       #sTimerLoadGripperOpened(IN := #sCurrent_Step_NB = 90 AND #iLoadGripperOpened,
                                PT := T#200ms);

       // Timer between approach and Load position
       #sTimerAfterApproach(IN := #sCurrent_Step_NB = 75 AND #iAxisW_FixtApproachPos,
                            PT := T#100ms);
   END_REGION

   REGION Sequence Function
       CASE #sCurrent_Step_NB OF
           #S00_INIT:
               REGION S00 INIT
                   #sCheck_Step_Condition := TRUE;
               END_REGION
           #S10_CHECK_FIXTURE_LOAD_OPTION:
               REGION S10_CHECK_FIXTURE_LOAD_OPTION
                   #sCheck_Step_Condition := TRUE;
               END_REGION
           #S20_AXIS_W_TO_FIXTURE_SAFE_POS_START_REQ:
               REGION S20_AXIS_W_TO_FIXTURE_SAFE_POS_START_REQ
                   #sAxisW_StartReq := NOT #iAxisW_FixtSafePos;
                   #sAxisW_PosSetPoint := LREAL_TO_REAL(#iAxisW_FixtSafePosSetPoint);
                   #sCheck_Step_Condition := TRUE;
               END_REGION
           #S30_AXIS_W_TO_FIXTURE_SAFE_POS_REACHED:
               REGION S30_AXIS_W_TO_FIXTURE_SAFE_POS_REACHED
                   #sCheck_Step_Condition := TRUE;
               END_REGION
           #S40_AXIS_V_TO_FIXTURE_LOAD_POS_START_REQ:
               REGION S40_AXIS_V_TO_FIXTURE_LOAD_POS_START_REQ
                   #sAxisV_StartReq := NOT #iAxisV_FixtLoadPos;
                   #sAxisV_PosSetPoint := LREAL_TO_REAL(#iAxisV_FixtLoadPosSetPoint);
                   #sCheck_Step_Condition := TRUE;
               END_REGION
           #S50_AXIS_V_TO_FIXTURE_LOAD_POS_REACHED:
               REGION S50_AXIS_V_TO_FIXTURE_LOAD_POS_REACHED
                   #sCheck_Step_Condition := TRUE;
               END_REGION
           #S60_OPEN_FIXTURE:
               REGION S60_OPEN_FIXTURE
                   #sFixtureOpenReq := TRUE;
                   IF #sTimerFixtureOpened.Q THEN
                       #sCheck_Step_Condition := TRUE;
                   END_IF;
               END_REGION


           #S70_AXIS_W_TO_FIXTURE_APPROACH_POS_START_REQ:
               REGION S70_AXIS_W_TO_FIXTURE_APPROACH_POS_START_REQ
                   #sAxisW_StartReq := NOT #iAxisW_FixtApproachPos;
                   #sAxisW_PosSetPoint := LREAL_TO_REAL(#iAxisW_FixtApproachPosSetPoint);
                   #sCheck_Step_Condition := TRUE;
               END_REGION
           #S75_AXIS_W_TO_FIXTURE_APPROACH_POS_REACHED:
               REGION S75_AXIS_W_TO_FIXTURE_APPROACH_POS_REACHED
                   IF #sTimerAfterApproach.Q THEN
                       #sCheck_Step_Condition := TRUE;
                   END_IF;
               END_REGION


           #S80_AXIS_W_TO_FIXTURE_LOAD_POS_START_REQ:
               REGION #S80_AXIS_W_TO_FIXTURE_LOAD_POS_START_REQ
                   #sAxisW_StartReq := NOT #iAxisW_FixtLoadPos;
                   #sAxisW_PosSetPoint := LREAL_TO_REAL(#iAxisW_FixtLoadPosSetPoint);
                   #sCheck_Step_Condition := TRUE;
               END_REGION
           #S85_AXIS_W_TO_FIXTURE_LOAD_POS_REACHED:
               REGION #S85_AXIS_W_TO_FIXTURE_LOAD_POS_REACHED
                   #sCheck_Step_Condition := TRUE;
               END_REGION
           #S90_OPEN_LOAD_GRIPPER:
               REGION S90_OPEN_LOAD_GRIPPER
                   #sLoadGripperOpenReq := TRUE;
                   IF #sTimerLoadGripperOpened.Q THEN
                       #sCheck_Step_Condition := TRUE;
                   END_IF;
               END_REGION
           #S95_VACUUM_START:
               REGION S95_VACUUM_START
                   #sVacuumStartReq := TRUE;
                   #sCheck_Step_Condition := TRUE;
               END_REGION
           #S100_AXIS_W_TO_FIXTURE_SAFE_POS_START_REQ:
               REGION S100_AXIS_W_TO_FIXTURE_SAFE_POS_START_REQ
                   #sAxisW_StartReq := NOT #iAxisW_FixtSafePos;
                   #sAxisW_PosSetPoint := LREAL_TO_REAL(#iAxisW_FixtSafePosSetPoint);
                   #sCheck_Step_Condition := TRUE;
               END_REGION
           #S110_AXIS_W_TO_FIXTURE_SAFE_POS_REACHED:
               REGION S110_AXIS_W_TO_FIXTURE_SAFE_POS_REACHED
                   #sCheck_Step_Condition := TRUE;
               END_REGION
           #S120_CLOSE_FIXTURE:
               REGION S120_CLOSE_FIXTURE
                   #sFixtureCloseReq := TRUE;
                   IF #sTimerFixtureClosed.Q THEN
                       #sCheck_Step_Condition := TRUE;
                   END_IF;
               END_REGION
           #S195_JOB_DONE:
               REGION S195_JOB_DONE
                   #sInterface.JobDone := TRUE;
                   #sCheck_Step_Condition := TRUE;
               END_REGION
           ELSE:
               #sInterface.Error := TRUE;
       END_CASE;
   END_REGION

   REGION Sequence Next Step Condition
       IF #sCheck_Step_Condition THEN
           CASE #sCurrent_Step_NB OF
               #S00_INIT:
                   REGION S00_INIT
                       IF #sInterface.SequenceReleased AND #iJobReq THEN
                           #sCurrent_Step_NB := #S10_CHECK_FIXTURE_LOAD_OPTION;
                           #sInterface.SequenceRun := TRUE;
                           #sCheck_Step_Condition := FALSE;
                       ELSE
                           #sInterface.SequenceRun := FALSE;
                       END_IF;
                   END_REGION
               #S10_CHECK_FIXTURE_LOAD_OPTION:
                   REGION S10_CHECK_FIXTURE_LOAD_OPTION
                       IF #sInterface.SequenceReleased AND #sStepForward AND NOT "DB_LoaderOptions".Fixture.LoadingDisabled THEN
                           #sCurrent_Step_NB := #S20_AXIS_W_TO_FIXTURE_SAFE_POS_START_REQ;
                           #sCheck_Step_Condition := FALSE;
                       ELSIF #sInterface.SequenceReleased AND #sStepForward AND "DB_LoaderOptions".Fixture.LoadingDisabled THEN
                           #sCurrent_Step_NB := #S195_JOB_DONE;
                           #sCheck_Step_Condition := FALSE;
                       END_IF;
                   END_REGION
               #S20_AXIS_W_TO_FIXTURE_SAFE_POS_START_REQ:
                   REGION S20_AXIS_W_TO_FIXTURE_SAFE_POS_START_REQ
                       IF #sInterface.SequenceReleased AND #sStepForward AND (#iAxisW_Moving OR #iAxisW_FixtSafePos) THEN
                           #sCurrent_Step_NB := #S30_AXIS_W_TO_FIXTURE_SAFE_POS_REACHED;
                           #sCheck_Step_Condition := FALSE;
                       END_IF;
                   END_REGION
               #S30_AXIS_W_TO_FIXTURE_SAFE_POS_REACHED:
                   REGION S30_AXIS_W_TO_FIXTURE_SAFE_POS_REACHED
                       IF #sInterface.SequenceReleased AND #sStepForward AND NOT #sAxisW_StartReq AND #iAxisW_FixtSafePos THEN
                           #sCurrent_Step_NB := #S40_AXIS_V_TO_FIXTURE_LOAD_POS_START_REQ;
                           #sCheck_Step_Condition := FALSE;
                       END_IF;
                   END_REGION
               #S40_AXIS_V_TO_FIXTURE_LOAD_POS_START_REQ:
                   REGION S40_AXIS_V_TO_FIXTURE_LOAD_POS_START_REQ
                       IF #sInterface.SequenceReleased AND #sStepForward AND (#iAxisV_Moving OR #iAxisV_FixtLoadPos) THEN
                           #sCurrent_Step_NB := #S50_AXIS_V_TO_FIXTURE_LOAD_POS_REACHED;
                           #sCheck_Step_Condition := FALSE;
                       END_IF;
                   END_REGION
               #S50_AXIS_V_TO_FIXTURE_LOAD_POS_REACHED:
                   REGION S50_AXIS_V_TO_FIXTURE_LOAD_POS_REACHED
                       IF #sInterface.SequenceReleased AND #sStepForward AND NOT #sAxisV_StartReq AND #iAxisV_FixtLoadPos THEN
                           #sCurrent_Step_NB := #S60_OPEN_FIXTURE;
                           #sCheck_Step_Condition := FALSE;
                       END_IF;
                   END_REGION
               #S60_OPEN_FIXTURE:
                   REGION S60_OPEN_FIXTURE
                       IF #sInterface.SequenceReleased AND #sStepForward AND #iFixtureOpened THEN
                           #sCurrent_Step_NB := #S70_AXIS_W_TO_FIXTURE_APPROACH_POS_START_REQ;
                           #sCheck_Step_Condition := FALSE;
                       END_IF;
                   END_REGION
               #S70_AXIS_W_TO_FIXTURE_APPROACH_POS_START_REQ:
                   REGION S70_AXIS_W_TO_FIXTURE_APPROACH_POS_START_REQ
                       IF #sInterface.SequenceReleased AND #sStepForward AND (#iAxisW_Moving OR #iAxisW_FixtApproachPos) THEN
                           #sCurrent_Step_NB := #S75_AXIS_W_TO_FIXTURE_APPROACH_POS_REACHED;
                           #sCheck_Step_Condition := FALSE;
                       END_IF;
                   END_REGION
               #S75_AXIS_W_TO_FIXTURE_APPROACH_POS_REACHED:
                   REGION S75_AXIS_W_TO_FIXTURE_APPROACH_POS_REACHED
                       IF #sInterface.SequenceReleased AND #sStepForward AND NOT #sAxisW_StartReq AND #iAxisW_FixtApproachPos THEN
                           #sCurrent_Step_NB := #S80_AXIS_W_TO_FIXTURE_LOAD_POS_START_REQ;
                           #sCheck_Step_Condition := FALSE;
                       END_IF;
                   END_REGION

               #S80_AXIS_W_TO_FIXTURE_LOAD_POS_START_REQ:
                   REGION S80_AXIS_W_TO_FIXTURE_LOAD_POS_START_REQ
                       IF #sInterface.SequenceReleased AND #sStepForward AND (#iAxisW_Moving OR #iAxisW_FixtLoadPos) THEN
                           #sCurrent_Step_NB := #S85_AXIS_W_TO_FIXTURE_LOAD_POS_REACHED;
                           #sCheck_Step_Condition := FALSE;
                       END_IF;
                   END_REGION
               #S85_AXIS_W_TO_FIXTURE_LOAD_POS_REACHED:
                   REGION S85_AXIS_W_TO_FIXTURE_LOAD_POS_REACHED
                       IF #sInterface.SequenceReleased AND #sStepForward AND NOT #sAxisW_StartReq AND #iAxisW_FixtLoadPos THEN
                           #sCurrent_Step_NB := #S90_OPEN_LOAD_GRIPPER;
                           #sCheck_Step_Condition := FALSE;
                       END_IF;
                   END_REGION


               #S90_OPEN_LOAD_GRIPPER:
                   REGION S90_OPEN_LOAD_GRIPPER
                       IF #sInterface.SequenceReleased AND #sStepForward AND #iLoadGripperOpened THEN
                           #sCurrent_Step_NB := #S95_VACUUM_START;
                           #sCheck_Step_Condition := FALSE;
                       END_IF;
                   END_REGION
               #S95_VACUUM_START:
                   REGION S95_VACUUM_START
                       IF #sInterface.SequenceReleased AND #sStepForward AND TRUE THEN
                           #sCurrent_Step_NB := #S100_AXIS_W_TO_FIXTURE_SAFE_POS_START_REQ;
                           #sCheck_Step_Condition := FALSE;
                       END_IF;
                   END_REGION
               #S100_AXIS_W_TO_FIXTURE_SAFE_POS_START_REQ:
                   REGION S100_AXIS_W_TO_FIXTURE_SAFE_POS_START_REQ
                       IF #sInterface.SequenceReleased AND #sStepForward AND (#iAxisW_Moving OR #iAxisW_FixtSafePos) THEN
                           #sCurrent_Step_NB := #S110_AXIS_W_TO_FIXTURE_SAFE_POS_REACHED;
                           #sCheck_Step_Condition := FALSE;
                       END_IF;
                   END_REGION
               #S110_AXIS_W_TO_FIXTURE_SAFE_POS_REACHED:
                   REGION S110_AXIS_W_TO_FIXTURE_SAFE_POS_REACHED
                       IF #sInterface.SequenceReleased AND #sStepForward AND NOT #sAxisW_StartReq AND #iAxisW_FixtSafePos THEN
                           #sCurrent_Step_NB := #S120_CLOSE_FIXTURE;
                           #sCheck_Step_Condition := FALSE;
                       END_IF;
                   END_REGION
               #S120_CLOSE_FIXTURE:
                   REGION S120_CLOSE_FIXTURE
                       IF #sInterface.SequenceReleased AND #sStepForward AND #iFixtureClosed THEN
                           #sCurrent_Step_NB := #S195_JOB_DONE;
                           #sCheck_Step_Condition := FALSE;
                       END_IF;
                   END_REGION
               #S195_JOB_DONE:
                   REGION S195_JOB_DONE
                       IF NOT #iJobReq THEN
                           #sCurrent_Step_NB := #S00_INIT;
                           #sCheck_Step_Condition := FALSE;
                           #sInterface.JobDone := FALSE;
                       END_IF;
                   END_REGION
               ELSE
                   #sInterface.Error := TRUE;
           END_CASE;
       END_IF;
   END_REGION

   REGION Outputs Update
       #oAxisV_StartReq := #sAxisV_StartReq;
       #oAxisV_PosSetPoint := #sAxisV_PosSetPoint;
       #oAxisW_StartReq := #sAxisW_StartReq;
       #oAxisW_PosSetPoint := #sAxisW_PosSetPoint;
       #oFixtureOpenReq := #sFixtureOpenReq;
       #oFixtureCloseReq := #sFixtureCloseReq;
       #oLoadGripperOpenReq := #sLoadGripperOpenReq;
       #oVacuumStartReq := #sVacuumStartReq;
   END_REGION

   REGION Steps - Date and Time History
       IF #sHistory.Activation THEN
           IF #sHistory.Steps[0] <> #sCurrent_Step_NB THEN
               FOR #tIndex := 98 TO 0 BY -1 DO
                   #sHistory.Steps[#tIndex + 1] := #sHistory.Steps[#tIndex];
                   #sHistory.Date_Time[#tIndex + 1] := #sHistory.Date_Time[#tIndex];
               END_FOR;
               #sHistory.Steps[0] := #sCurrent_Step_NB;
               #sHistory.Date_Time[0] := #iPLC_DateAndTime;
           END_IF;
       END_IF;
   END_REGION

   REGION Steps Text
       #StepText(iErrorCode := #sCurrent_Step_NB,
                 oErrorText => #StepText.oErrorText);
   END_REGION
END_FUNCTION_BLOCK

FUNCTION_BLOCK "FB_FixtureBlowing"   // FB68, SCL
{ S7_Optimized_Access := 'TRUE' }
// stored: AutoNumber false, MemoryReserve 100, SetENOAutomatically false
   VAR_INPUT
      iStartSeqCond : Bool;   // Start Sequence Conditions
      iJobReq : Bool;   // Job Request - From Main
      iFixtureOpened : Bool;
      iAxisV_FixtBlowingPos : Bool;
      iAxisV_FixtBlowingPosSetPoint : LReal;
      iAxisW_FixtSafePos : Bool;
      iAxisW_FixtSafePosSetPoint : LReal;
      iAxisW_FixtBlowPos : Bool;
      iAxisW_FixtBlowPosSetPoint : LReal;
      iAxisV_Moving : Bool;   // Shuttle is moving
      iAxisV_InPos : Bool;
      iAxisW_Moving { ExternalAccessible := 'False'; ExternalVisible := 'False'; ExternalWritable := 'False'} : Bool;   // Shuttle is moving
      iAxisW_InPos : Bool;
      iBlowingTime : Time;
      iPLC_DateAndTime : DTL;
      iStepPause : Bool;
   END_VAR
   VAR_OUTPUT
      oFixtureOpenReq : Bool;
      oAxisV_StartReq : Bool;
      oAxisV_PosSetPoint : Real;
      oAxisW_StartReq : Bool;
      oAxisW_PosSetPoint : Real;
      oBlowingReq : Bool;
   END_VAR
   VAR
      sCurrent_Step_NB : Int;   // Active Step Number
      sCheck_Step_Condition : Bool;
      sOneStepForward : Bool;
      sRTOneStepForward : R_TRIG;
      sOneStepMode { S7_SetPoint := 'True'} : Bool;
      sStepForward : Bool;
      sInterface : "UDT_SequenceInterface";
      sFixtureOpenReq { S7_SetPoint := 'True'} : Bool;
      sAxisV_StartReq : Bool;
      sAxisV_PosSetPoint : Real;
      sAxisW_StartReq : Bool;
      sAxisW_PosSetPoint : Real;
      sBlowingReq : Bool;   // Drilled Part To Unload - From FB_Position
      sBlowingTimerStart : Bool;
      sBlowingTimer : TP_TIME;
      sFT_BlowingTimer { S7_SetPoint := 'True'} : F_TRIG;
      sTimerFixtureOpened : TON_TIME;
      sHistory : Struct
         Activation : Bool;
         Steps : Array[0..99] of Int;
         Date_Time : Array[0..99] of DTL;
      END_STRUCT;
      StepText : "FB_GetTextErrorCode";
   END_VAR
   VAR_TEMP
      tIndex : Int;   // Index
   END_VAR
   VAR CONSTANT
      S00_INIT : Int := 0;
      S10_CHECK_FIXTURE_BLOW_OPTION : Int := 10;
      S20_AXIS_W_TO_FIXTURE_SAFE_POS_START_REQ : Int := 20;
      S30_AXIS_W_TO_FIXTURE_SAFE_POS_REACHED : Int := 30;
      S40_AXIS_V_TO_FIXTURE_BLOW_POS_START_REQ : Int := 40;
      S50_AXIS_V_TO_FIXTURE_BLOW_POS_REACHED : Int := 50;
      S60_OPEN_FIXTURE : Int := 60;
      S70_AXIS_W_TO_FIXTURE_BLOW_POS_START_REQ : Int := 70;
      S80_AXIS_W_TO_FIXTURE_BLOW_POS_REACHED : Int := 80;
      S90_BLOWING_TIMER_START_REQ : Int := 90;
      S100_AXIS_W_TO_FIXTURE_SAFE_POS_START_REQ : Int := 100;
      S110_AXIS_W_TO_FIXTURE_SAFE_POS_REACHED : Int := 110;
      S195_JOB_DONE : Int := 195;
   END_VAR
   // StepText.sCode_error[0].ErrorCode := 0;
   // StepText.sCode_error[1].ErrorCode := 10;
   // StepText.sCode_error[2].ErrorCode := 20;
   // StepText.sCode_error[3].ErrorCode := 30;
   // StepText.sCode_error[4].ErrorCode := 40;
   // StepText.sCode_error[5].ErrorCode := 50;
   // StepText.sCode_error[6].ErrorCode := 60;
   // StepText.sCode_error[7].ErrorCode := 70;
   // StepText.sCode_error[8].ErrorCode := 80;
   // StepText.sCode_error[9].ErrorCode := 90;
   // StepText.sCode_error[10].ErrorCode := 95;
BEGIN
   REGION Description header 
       //==================================================================================
       // POSALUX Swiss SA / (C) Copyright 2026
       //----------------------------------------------------------------------------------
       // Title: FB_FixtureBlowing
       // Comment/Function: 
       // Author: Fabien WALDT
       // Engineering: TIA Portal v20
       //----------------------------------------------------------------------------------
       // Change log table:
       // Version  | Date     | Expert in charge | Changes applied
       // ---------|----------|------------------|-----------------------------------------
       // 00.00.01 | 20260122 | WFA              | First released version
       // =================================================================================
   END_REGION

   REGION Define condition to start
       IF #iStartSeqCond THEN
           #sInterface.SequenceReleased := TRUE;
       ELSE
           // Standard sequencer controls
           #sInterface.SequenceReleased := FALSE;
           #sCurrent_Step_NB := #S00_INIT;
           #sInterface.SequenceRun := FALSE;
           #sInterface.JobDone := FALSE;
           #sCheck_Step_Condition := FALSE;

           // Dedicated sequencer controls
           #sAxisV_StartReq := FALSE;
           #sAxisV_PosSetPoint := 0.0;
           #sAxisW_StartReq := FALSE;
           #sAxisW_PosSetPoint := 0.0;
           #sFixtureOpenReq := FALSE;
           #sBlowingReq := FALSE;
           #sBlowingTimerStart := FALSE;

           // Add specifics controls 
       END_IF;

       // Reset interface error
       IF #sInterface.Reset THEN
           #sInterface.Error := FALSE;
       END_IF;

       // Reset start when axis in position
       IF #iAxisV_InPos THEN
           #sAxisV_StartReq := FALSE;
       END_IF;
       IF #iAxisW_InPos THEN
           #sAxisW_StartReq := FALSE;
       END_IF;

       // One step forward
       #sRTOneStepForward.CLK := #sOneStepForward;
       #sRTOneStepForward();
       #sStepForward := (NOT #sOneStepMode OR (#sOneStepMode AND #sRTOneStepForward.Q)) AND NOT #iStepPause;
       #sOneStepForward := FALSE;

       // Blowing Timer
       #sBlowingTimer(IN := #sBlowingTimerStart,
                      PT := #iBlowingTime);

       #sFT_BlowingTimer(CLK := #sBlowingTimer.Q);

       #sBlowingReq := #sBlowingTimer.Q
       OR #sCurrent_Step_NB = 70
       OR #sCurrent_Step_NB = 80;
       // Action only true in dedicated steps
       #sFixtureOpenReq := FALSE;
       #sBlowingTimerStart := FALSE;

       // Step Timer
       #sTimerFixtureOpened(IN := #sCurrent_Step_NB = 60 AND #iFixtureOpened,
                            PT := T#1000ms);
   END_REGION

   REGION Sequence Function
       CASE #sCurrent_Step_NB OF
           #S00_INIT:
               REGION S00 INIT
                   #sCheck_Step_Condition := TRUE;
               END_REGION
           #S10_CHECK_FIXTURE_BLOW_OPTION:
               REGION S10_CHECK_FIXTURE_BLOW_OPTION
                   #sCheck_Step_Condition := TRUE;
               END_REGION
           #S20_AXIS_W_TO_FIXTURE_SAFE_POS_START_REQ:
               REGION S20_AXIS_W_TO_FIXTURE_SAFE_POS_START_REQ
                   #sAxisW_StartReq := NOT #iAxisW_FixtSafePos;
                   #sAxisW_PosSetPoint := LREAL_TO_REAL(#iAxisW_FixtSafePosSetPoint);
                   #sCheck_Step_Condition := TRUE;
               END_REGION
           #S30_AXIS_W_TO_FIXTURE_SAFE_POS_REACHED:
               REGION S30_AXIS_W_TO_FIXTURE_SAFE_POS_REACHED
                   #sCheck_Step_Condition := TRUE;
               END_REGION
           #S40_AXIS_V_TO_FIXTURE_BLOW_POS_START_REQ:
               REGION S40_AXIS_V_TO_FIXTURE_BLOW_POS_START_REQ
                   #sAxisV_StartReq := NOT #iAxisV_FixtBlowingPos;
                   #sAxisV_PosSetPoint := LREAL_TO_REAL(#iAxisV_FixtBlowingPosSetPoint);
                   #sCheck_Step_Condition := TRUE;
               END_REGION
           #S50_AXIS_V_TO_FIXTURE_BLOW_POS_REACHED:
               REGION S50_AXIS_V_TO_FIXTURE_BLOW_POS_REACHED
                   #sCheck_Step_Condition := TRUE;
               END_REGION
           #S60_OPEN_FIXTURE:
               REGION S60_OPEN_FIXTURE
                   #sFixtureOpenReq := TRUE;
                   IF #sTimerFixtureOpened.Q THEN
                       #sCheck_Step_Condition := TRUE;
                   END_IF;
               END_REGION
           #S70_AXIS_W_TO_FIXTURE_BLOW_POS_START_REQ:
               REGION S70_AXIS_W_TO_FIXTURE_BLOW_POS_START_REQ
                   #sAxisW_StartReq := NOT #iAxisW_FixtBlowPos;
                   #sAxisW_PosSetPoint := LREAL_TO_REAL(#iAxisW_FixtBlowPosSetPoint);
                   #sCheck_Step_Condition := TRUE;
               END_REGION
           #S80_AXIS_W_TO_FIXTURE_BLOW_POS_REACHED:
               REGION S80_AXIS_W_TO_FIXTURE_BLOW_POS_REACHED
                   #sCheck_Step_Condition := TRUE;
               END_REGION
           #S90_BLOWING_TIMER_START_REQ:
               REGION S90_BLOWING_TIMER_START_REQ
                   #sBlowingTimerStart := TRUE;
                   #sCheck_Step_Condition := TRUE;
               END_REGION
           #S100_AXIS_W_TO_FIXTURE_SAFE_POS_START_REQ:
               REGION S100_AXIS_W_TO_FIXTURE_SAFE_POS_START_REQ
                   #sAxisW_StartReq := NOT #iAxisW_FixtSafePos;
                   #sAxisW_PosSetPoint := LREAL_TO_REAL(#iAxisW_FixtSafePosSetPoint);
                   #sCheck_Step_Condition := TRUE;
               END_REGION
           #S110_AXIS_W_TO_FIXTURE_SAFE_POS_REACHED:
               REGION S110_AXIS_W_TO_FIXTURE_SAFE_POS_REACHED
                   #sCheck_Step_Condition := TRUE;
               END_REGION
           #S195_JOB_DONE:
               REGION S195_JOB_DONE
                   #sInterface.JobDone := TRUE;
                   #sCheck_Step_Condition := TRUE;
               END_REGION
           ELSE:
               #sInterface.Error := TRUE;
       END_CASE;
   END_REGION

   REGION Sequence Next Step Condition
       IF #sCheck_Step_Condition THEN
           CASE #sCurrent_Step_NB OF
               #S00_INIT:
                   REGION S00_INIT
                       IF #sInterface.SequenceReleased AND #iJobReq THEN
                           #sCurrent_Step_NB := #S10_CHECK_FIXTURE_BLOW_OPTION;
                           #sInterface.SequenceRun := TRUE;
                           #sCheck_Step_Condition := FALSE;
                       ELSE
                           #sInterface.SequenceRun := FALSE;
                       END_IF;
                   END_REGION
               #S10_CHECK_FIXTURE_BLOW_OPTION:
                   REGION S10_CHECK_FIXTURE_UNLOAD_OPTION
                       IF #sInterface.SequenceReleased AND #sStepForward AND NOT "DB_LoaderOptions".Fixture.BlowingDisabled  THEN
                           #sCurrent_Step_NB := #S20_AXIS_W_TO_FIXTURE_SAFE_POS_START_REQ;
                           #sCheck_Step_Condition := FALSE;
                       ELSIF #sInterface.SequenceReleased AND #sStepForward AND "DB_LoaderOptions".Fixture.BlowingDisabled THEN
                           #sCurrent_Step_NB := #S195_JOB_DONE;
                           #sCheck_Step_Condition := FALSE;
                       END_IF;
                   END_REGION
               #S20_AXIS_W_TO_FIXTURE_SAFE_POS_START_REQ:
                   REGION S20_AXIS_W_TO_FIXTURE_SAFE_POS_START_REQ
                       IF #sInterface.SequenceReleased AND #sStepForward AND (#iAxisW_Moving OR #iAxisW_FixtSafePos) THEN
                           #sCurrent_Step_NB := #S30_AXIS_W_TO_FIXTURE_SAFE_POS_REACHED;
                           #sCheck_Step_Condition := FALSE;
                       END_IF;
                   END_REGION
               #S30_AXIS_W_TO_FIXTURE_SAFE_POS_REACHED:
                   REGION S30_AXIS_W_TO_FIXTURE_SAFE_POS_REACHED
                       IF #sInterface.SequenceReleased AND #sStepForward AND NOT #sAxisW_StartReq AND #iAxisW_FixtSafePos THEN
                           #sCurrent_Step_NB := #S40_AXIS_V_TO_FIXTURE_BLOW_POS_START_REQ;
                           #sCheck_Step_Condition := FALSE;
                       END_IF;
                   END_REGION
               #S40_AXIS_V_TO_FIXTURE_BLOW_POS_START_REQ:
                   REGION S40_AXIS_V_TO_FIXTURE_BLOW_POS_START_REQ
                       IF #sInterface.SequenceReleased AND #sStepForward AND (#iAxisV_Moving OR #iAxisV_FixtBlowingPos) THEN
                           #sCurrent_Step_NB := #S50_AXIS_V_TO_FIXTURE_BLOW_POS_REACHED;
                           #sCheck_Step_Condition := FALSE;
                       END_IF;
                   END_REGION
               #S50_AXIS_V_TO_FIXTURE_BLOW_POS_REACHED:
                   REGION S50_AXIS_V_TO_FIXTURE_BLOW_POS_REACHED
                       IF #sInterface.SequenceReleased AND #sStepForward AND NOT #sAxisV_StartReq AND #iAxisV_FixtBlowingPos THEN
                           #sCurrent_Step_NB := #S60_OPEN_FIXTURE;
                           #sCheck_Step_Condition := FALSE;
                       END_IF;
                   END_REGION
               #S60_OPEN_FIXTURE:
                   REGION S60_OPEN_FIXTURE
                       IF #sInterface.SequenceReleased AND #sStepForward AND #iFixtureOpened THEN
                           #sCurrent_Step_NB := #S70_AXIS_W_TO_FIXTURE_BLOW_POS_START_REQ;
                           #sCheck_Step_Condition := FALSE;
                       END_IF;
                   END_REGION
               #S70_AXIS_W_TO_FIXTURE_BLOW_POS_START_REQ:
                   REGION S70_AXIS_W_TO_FIXTURE_BLOW_POS_START_REQ
                       IF #sInterface.SequenceReleased AND #sStepForward AND (#iAxisW_Moving OR #iAxisW_FixtBlowPos) THEN
                           #sCurrent_Step_NB := #S80_AXIS_W_TO_FIXTURE_BLOW_POS_REACHED;
                           #sCheck_Step_Condition := FALSE;
                       END_IF;
                   END_REGION
               #S80_AXIS_W_TO_FIXTURE_BLOW_POS_REACHED:
                   REGION S80_AXIS_W_TO_FIXTURE_BLOW_POS_REACHED
                       IF #sInterface.SequenceReleased AND #sStepForward AND NOT #sAxisW_StartReq AND #iAxisW_FixtBlowPos THEN
                           #sCurrent_Step_NB := #S90_BLOWING_TIMER_START_REQ;
                           #sCheck_Step_Condition := FALSE;
                       END_IF;
                   END_REGION
               #S90_BLOWING_TIMER_START_REQ:
                   REGION S90_BLOWING_TIMER_START_REQ
                       IF #sInterface.SequenceReleased AND #sStepForward AND #sFT_BlowingTimer.Q THEN
                           #sCurrent_Step_NB := #S100_AXIS_W_TO_FIXTURE_SAFE_POS_START_REQ;
                           #sCheck_Step_Condition := FALSE;
                       END_IF;
                   END_REGION
               #S100_AXIS_W_TO_FIXTURE_SAFE_POS_START_REQ:
                   REGION S100_AXIS_W_TO_FIXTURE_SAFE_POS_START_REQ
                       IF #sInterface.SequenceReleased AND #sStepForward AND (#iAxisW_Moving OR #iAxisW_FixtSafePos) THEN
                           #sCurrent_Step_NB := #S110_AXIS_W_TO_FIXTURE_SAFE_POS_REACHED;
                           #sCheck_Step_Condition := FALSE;
                       END_IF;
                   END_REGION
               #S110_AXIS_W_TO_FIXTURE_SAFE_POS_REACHED:
                   REGION S110_AXIS_W_TO_FIXTURE_SAFE_POS_REACHED
                       IF #sInterface.SequenceReleased AND #sStepForward AND NOT #sAxisW_StartReq AND #iAxisW_FixtSafePos THEN
                           #sCurrent_Step_NB := #S195_JOB_DONE;
                           #sCheck_Step_Condition := FALSE;
                       END_IF;
                   END_REGION
               #S195_JOB_DONE:
                   REGION S195_JOB_DONE
                       IF NOT #iJobReq THEN
                           #sCurrent_Step_NB := #S00_INIT;
                           #sCheck_Step_Condition := FALSE;
                           #sInterface.JobDone := FALSE;
                       END_IF;
                   END_REGION
               ELSE
                   #sInterface.Error := TRUE;
           END_CASE;
       END_IF;
   END_REGION

   REGION Outputs Update
       #oAxisV_StartReq := #sAxisV_StartReq;
       #oAxisV_PosSetPoint := #sAxisV_PosSetPoint;
       #oAxisW_StartReq := #sAxisW_StartReq;
       #oAxisW_PosSetPoint := #sAxisW_PosSetPoint;
       #oFixtureOpenReq := #sFixtureOpenReq;
       #oBlowingReq := #sBlowingReq;
   END_REGION

   REGION Steps - Date and Time History
       IF #sHistory.Activation THEN
           IF #sHistory.Steps[0] <> #sCurrent_Step_NB THEN
               FOR #tIndex := 98 TO 0 BY -1 DO
                   #sHistory.Steps[#tIndex + 1] := #sHistory.Steps[#tIndex];
                   #sHistory.Date_Time[#tIndex + 1] := #sHistory.Date_Time[#tIndex];
               END_FOR;
               #sHistory.Steps[0] := #sCurrent_Step_NB;
               #sHistory.Date_Time[0] := #iPLC_DateAndTime;
           END_IF;
       END_IF;
   END_REGION

   REGION Steps Text
       #StepText(iErrorCode := #sCurrent_Step_NB,
                 oErrorText => #StepText.oErrorText);
   END_REGION
END_FUNCTION_BLOCK

FUNCTION_BLOCK "FB_FixtureRelease"   // FB70, SCL
{ S7_Optimized_Access := 'TRUE' }
// stored: AutoNumber false, MemoryReserve 100, SetENOAutomatically false
   VAR_INPUT
      iStartSeqCond : Bool;   // Start Sequence Conditions
      iJobReq : Bool;   // Job Request - From Main
      iAxisV_SafePos : Bool;
      iAxisV_SafePosSetPoint : LReal;
      iAxisW_FixtSafePos : Bool;
      iAxisW_FixtSafePosSetPoint : LReal;
      iAxisV_Moving : Bool;   // Shuttle is moving
      iAxisV_InPos : Bool;
      iAxisW_Moving { ExternalAccessible := 'False'; ExternalVisible := 'False'; ExternalWritable := 'False'} : Bool;   // Shuttle is moving
      iAxisW_InPos : Bool;
      iPLC_DateAndTime : DTL;
      iStepPause : Bool;
   END_VAR
   VAR_OUTPUT
      oAxisV_StartReq : Bool;
      oAxisV_PosSetPoint : Real;
      oAxisW_StartReq : Bool;
      oAxisW_PosSetPoint : Real;
   END_VAR
   VAR
      sCurrent_Step_NB : Int;   // Active Step Number
      sCheck_Step_Condition : Bool;
      sOneStepForward : Bool;
      sRTOneStepForward : R_TRIG;
      sOneStepMode { S7_SetPoint := 'True'} : Bool;
      sStepForward : Bool;
      sInterface : "UDT_SequenceInterface";
      sAxisV_StartReq : Bool;
      sAxisV_PosSetPoint : Real;
      sAxisW_StartReq : Bool;
      sAxisW_PosSetPoint : Real;
      sHistory : Struct
         Activation : Bool;
         Steps : Array[0..99] of Int;
         Date_Time : Array[0..99] of DTL;
      END_STRUCT;
      StepText : "FB_GetTextErrorCode";
   END_VAR
   VAR_TEMP
      tIndex : Int;   // Index
   END_VAR
   VAR CONSTANT
      S00_INIT : Int := 0;
      S10_CHECK_FIXTURE_RELEASE_OPTION : Int := 10;
      S20_AXIS_W_TO_FIXTURE_SAFE_POS_START_REQ : Int := 20;
      S30_AXIS_W_TO_FIXTURE_SAFE_POS_REACHED : Int := 30;
      S40_AXIS_V_TO_SHUTTLE_SAFE_POS_START_REQ : Int := 40;
      S50_AXIS_V_TO_SHUTTLE_SAFE_POS_REACHED : Int := 50;
      S95_JOB_DONE : Int := 95;
   END_VAR
   // StepText.sCode_error[0].ErrorCode := 0;
   // StepText.sCode_error[1].ErrorCode := 10;
   // StepText.sCode_error[2].ErrorCode := 20;
   // StepText.sCode_error[3].ErrorCode := 30;
   // StepText.sCode_error[4].ErrorCode := 40;
   // StepText.sCode_error[5].ErrorCode := 50;
   // StepText.sCode_error[6].ErrorCode := 60;
   // StepText.sCode_error[7].ErrorCode := 70;
   // StepText.sCode_error[8].ErrorCode := 80;
   // StepText.sCode_error[9].ErrorCode := 90;
   // StepText.sCode_error[10].ErrorCode := 95;
BEGIN
   REGION Description header 
       //==================================================================================
       // POSALUX Swiss SA / (C) Copyright 2026
       //----------------------------------------------------------------------------------
       // Title: FB_FixtureRelease
       // Comment/Function: 
       // Author: Fabien WALDT
       // Engineering: TIA Portal v20
       //----------------------------------------------------------------------------------
       // Change log table:
       // Version  | Date     | Expert in charge | Changes applied
       // ---------|----------|------------------|-----------------------------------------
       // 00.00.01 | 20260122 | WFA              | First released version
       // =================================================================================
   END_REGION

   REGION Define condition to start
       IF #iStartSeqCond THEN
           #sInterface.SequenceReleased := TRUE;
       ELSE
           // Standard sequencer controls
           #sInterface.SequenceReleased := FALSE;
           #sCurrent_Step_NB := #S00_INIT;
           #sInterface.SequenceRun := FALSE;
           #sInterface.JobDone := FALSE;
           #sCheck_Step_Condition := FALSE;

           // Dedicated sequencer controls
           #sAxisV_StartReq := FALSE;
           #sAxisV_PosSetPoint := 0.0;
           #sAxisW_StartReq := FALSE;
           #sAxisW_PosSetPoint := 0.0;

           // Add specifics controls 
       END_IF;

       // Reset interface error
       IF #sInterface.Reset THEN
           #sInterface.Error := FALSE;
       END_IF;

       // Reset start when axis in position
       IF #iAxisV_InPos THEN
           #sAxisV_StartReq := FALSE;
       END_IF;
       IF #iAxisW_InPos THEN
           #sAxisW_StartReq := FALSE;
       END_IF;

       // One step forward
       #sRTOneStepForward.CLK := #sOneStepForward;
       #sRTOneStepForward();
       #sStepForward := (NOT #sOneStepMode OR (#sOneStepMode AND #sRTOneStepForward.Q)) AND NOT #iStepPause;
       #sOneStepForward := FALSE;

       // Action only true in dedicated steps

       // Step Timer

   END_REGION

   REGION Sequence Function
       CASE #sCurrent_Step_NB OF
           #S00_INIT:
               REGION S00 INIT
                   #sCheck_Step_Condition := TRUE;
               END_REGION
           #S10_CHECK_FIXTURE_RELEASE_OPTION:
               REGION S10_CHECK_FIXTURE_RELEASE_OPTION
                   #sCheck_Step_Condition := TRUE;
               END_REGION
           #S20_AXIS_W_TO_FIXTURE_SAFE_POS_START_REQ:
               REGION S20_AXIS_W_TO_FIXTURE_SAFE_POS_START_REQ
                   #sAxisW_StartReq := NOT #iAxisW_FixtSafePos;
                   #sAxisW_PosSetPoint := LREAL_TO_REAL(#iAxisW_FixtSafePosSetPoint);
                   #sCheck_Step_Condition := TRUE;
               END_REGION
           #S30_AXIS_W_TO_FIXTURE_SAFE_POS_REACHED:
               REGION S30_AXIS_W_TO_FIXTURE_SAFE_POS_REACHED
                   #sCheck_Step_Condition := TRUE;
               END_REGION
           #S40_AXIS_V_TO_SHUTTLE_SAFE_POS_START_REQ:
               REGION S40_AXIS_V_TO_SHUTTLE_SAFE_POS_START_REQ
                   #sAxisV_StartReq := NOT #iAxisV_SafePos;
                   #sAxisV_PosSetPoint := LREAL_TO_REAL(#iAxisV_SafePosSetPoint);
                   #sCheck_Step_Condition := TRUE;
               END_REGION
           #S50_AXIS_V_TO_SHUTTLE_SAFE_POS_REACHED:
               REGION S50_AXIS_V_TO_SHUTTLE_SAFE_POS_REACHED
                   #sCheck_Step_Condition := TRUE;
               END_REGION
           #S95_JOB_DONE:
               REGION S95_JOB_DONE
                   #sInterface.JobDone := TRUE;
                   #sCheck_Step_Condition := TRUE;
               END_REGION
           ELSE:
               #sInterface.Error := TRUE;
       END_CASE;
   END_REGION

   REGION Sequence Next Step Condition
       IF #sCheck_Step_Condition THEN
           CASE #sCurrent_Step_NB OF
               #S00_INIT:
                   REGION S00_INIT
                       IF #sInterface.SequenceReleased AND #iJobReq THEN
                           #sCurrent_Step_NB := #S10_CHECK_FIXTURE_RELEASE_OPTION;
                           #sInterface.SequenceRun := TRUE;
                           #sCheck_Step_Condition := FALSE;
                       ELSE
                           #sInterface.SequenceRun := FALSE;
                       END_IF;
                   END_REGION
               #S10_CHECK_FIXTURE_RELEASE_OPTION:
                   REGION S10_CHECK_FIXTURE_RELEASE_OPTION
                       IF #sInterface.SequenceReleased AND #sStepForward AND NOT "DB_LoaderOptions".Fixture.ReleaseDisabled  THEN
                           #sCurrent_Step_NB := #S20_AXIS_W_TO_FIXTURE_SAFE_POS_START_REQ;
                           #sCheck_Step_Condition := FALSE;
                       ELSIF #sInterface.SequenceReleased AND #sStepForward AND "DB_LoaderOptions".Fixture.ReleaseDisabled THEN
                           #sCurrent_Step_NB := #S95_JOB_DONE;
                           #sCheck_Step_Condition := FALSE;
                       END_IF;
                   END_REGION
               #S20_AXIS_W_TO_FIXTURE_SAFE_POS_START_REQ:
                   REGION S20_AXIS_W_TO_FIXTURE_SAFE_POS_START_REQ
                       IF #sInterface.SequenceReleased AND #sStepForward AND (#iAxisW_Moving OR #iAxisW_FixtSafePos) THEN
                           #sCurrent_Step_NB := #S30_AXIS_W_TO_FIXTURE_SAFE_POS_REACHED;
                           #sCheck_Step_Condition := FALSE;
                       END_IF;
                   END_REGION
               #S30_AXIS_W_TO_FIXTURE_SAFE_POS_REACHED:
                   REGION S30_AXIS_W_TO_FIXTURE_SAFE_POS_REACHED
                       IF #sInterface.SequenceReleased AND #sStepForward AND NOT #sAxisW_StartReq AND #iAxisW_FixtSafePos THEN
                           #sCurrent_Step_NB := #S40_AXIS_V_TO_SHUTTLE_SAFE_POS_START_REQ;
                           #sCheck_Step_Condition := FALSE;
                       END_IF;
                   END_REGION
               #S40_AXIS_V_TO_SHUTTLE_SAFE_POS_START_REQ:
                   REGION S40_AXIS_V_TO_SHUTTLE_SAFE_POS_START_REQ
                       IF #sInterface.SequenceReleased AND #sStepForward AND (#iAxisV_Moving OR #iAxisV_SafePos) THEN
                           #sCurrent_Step_NB := #S50_AXIS_V_TO_SHUTTLE_SAFE_POS_REACHED;
                           #sCheck_Step_Condition := FALSE;
                       END_IF;
                   END_REGION
               #S50_AXIS_V_TO_SHUTTLE_SAFE_POS_REACHED:
                   REGION S50_AXIS_V_TO_SHUTTLE_SAFE_POS_REACHED
                       IF #sInterface.SequenceReleased AND #sStepForward AND NOT #sAxisV_StartReq AND #iAxisV_SafePos THEN
                           #sCurrent_Step_NB := #S95_JOB_DONE;
                           #sCheck_Step_Condition := FALSE;
                       END_IF;
                   END_REGION
               #S95_JOB_DONE:
                   REGION S95_JOB_DONE
                       IF NOT #iJobReq THEN
                           #sCurrent_Step_NB := #S00_INIT;
                           #sCheck_Step_Condition := FALSE;
                           #sInterface.JobDone := FALSE;
                       END_IF;
                   END_REGION
               ELSE
                   #sInterface.Error := TRUE;
           END_CASE;
       END_IF;
   END_REGION

   REGION Outputs Update
       #oAxisV_StartReq := #sAxisV_StartReq;
       #oAxisV_PosSetPoint := #sAxisV_PosSetPoint;
       #oAxisW_StartReq := #sAxisW_StartReq;
       #oAxisW_PosSetPoint := #sAxisW_PosSetPoint;
   END_REGION

   REGION Steps - Date and Time History
       IF #sHistory.Activation THEN
           IF #sHistory.Steps[0] <> #sCurrent_Step_NB THEN
               FOR #tIndex := 98 TO 0 BY -1 DO
                   #sHistory.Steps[#tIndex + 1] := #sHistory.Steps[#tIndex];
                   #sHistory.Date_Time[#tIndex + 1] := #sHistory.Date_Time[#tIndex];
               END_FOR;
               #sHistory.Steps[0] := #sCurrent_Step_NB;
               #sHistory.Date_Time[0] := #iPLC_DateAndTime;
           END_IF;
       END_IF;
   END_REGION

   REGION Steps Text
       #StepText(iErrorCode := #sCurrent_Step_NB,
                 oErrorText => #StepText.oErrorText);
   END_REGION
END_FUNCTION_BLOCK

FUNCTION_BLOCK "FB_FixtureV_Init"   // FB77, SCL
{ S7_Optimized_Access := 'TRUE' }
// stored: AutoNumber false, MemoryReserve 100, SetENOAutomatically false
   VAR_INPUT
      iStartSeqCond : Bool;   // Start Sequence Conditions
      iJobReq : Bool;   // Job Request - From Main
      iAxisV_FixtSafePos : Bool;
      iAxisV_FixtSafePosSetPoint : LReal;
      iAxisV_Moving : Bool;   // Shuttle is moving
      iAxisV_InPos : Bool;
      iPLC_DateAndTime : DTL;
      iStepPause : Bool;
   END_VAR
   VAR_OUTPUT
      oAxisV_StartReq : Bool;
      oAxisV_PosSetPoint : Real;
   END_VAR
   VAR
      sCurrent_Step_NB : Int;   // Active Step Number
      sCheck_Step_Condition : Bool;
      sOneStepForward : Bool;
      sRTOneStepForward : R_TRIG;
      sOneStepMode { S7_SetPoint := 'True'} : Bool;
      sStepForward : Bool;
      sInterface : "UDT_SequenceInterface";
      sAxisV_StartReq : Bool;
      sAxisV_PosSetPoint : Real;
      sHistory : Struct
         Activation : Bool;
         Steps : Array[0..99] of Int;
         Date_Time : Array[0..99] of DTL;
      END_STRUCT;
      StepText : "FB_GetTextErrorCode";
   END_VAR
   VAR_TEMP
      tIndex : Int;   // Index
   END_VAR
   VAR CONSTANT
      S00_INIT : Int := 0;
      S10_CHECK_FIXTURE_RELEASE_OPTION : Int := 10;
      S20_AXIS_V_TO_FIXTURE_SAFE_POS_START_REQ : Int := 20;
      S30_AXIS_V_TO_FIXTURE_SAFE_POS_REACHED : Int := 30;
      S95_JOB_DONE : Int := 95;
   END_VAR
   // StepText.sCode_error[0].ErrorCode := 0;
   // StepText.sCode_error[1].ErrorCode := 10;
   // StepText.sCode_error[2].ErrorCode := 20;
   // StepText.sCode_error[3].ErrorCode := 30;
   // StepText.sCode_error[4].ErrorCode := 40;
   // StepText.sCode_error[5].ErrorCode := 50;
   // StepText.sCode_error[6].ErrorCode := 60;
   // StepText.sCode_error[7].ErrorCode := 70;
   // StepText.sCode_error[8].ErrorCode := 80;
   // StepText.sCode_error[9].ErrorCode := 90;
   // StepText.sCode_error[10].ErrorCode := 95;
BEGIN
   REGION Description header 
       //==================================================================================
       // POSALUX Swiss SA / (C) Copyright 2026
       //----------------------------------------------------------------------------------
       // Title: FB_FixtureV_Init
       // Comment/Function: 
       // Author: Fabien WALDT
       // Engineering: TIA Portal v20
       //----------------------------------------------------------------------------------
       // Change log table:
       // Version  | Date     | Expert in charge | Changes applied
       // ---------|----------|------------------|-----------------------------------------
       // 00.00.01 | 20260220 | WFA              | First released version
       // =================================================================================
   END_REGION

   REGION Define condition to start
       IF #iStartSeqCond THEN
           #sInterface.SequenceReleased := TRUE;
       ELSE
           // Standard sequencer controls
           #sInterface.SequenceReleased := FALSE;
           #sCurrent_Step_NB := #S00_INIT;
           #sInterface.SequenceRun := FALSE;
           #sInterface.JobDone := FALSE;
           #sCheck_Step_Condition := FALSE;

           // Dedicated sequencer controls
           #sAxisV_StartReq := FALSE;
           #sAxisV_PosSetPoint := 0.0;

           // Add specifics controls 
       END_IF;

       // Reset interface error
       IF #sInterface.Reset THEN
           #sInterface.Error := FALSE;
       END_IF;

       // Reset start when axis in position
       IF #iAxisV_InPos THEN
           #sAxisV_StartReq := FALSE;
       END_IF;

       // One step forward
       #sRTOneStepForward.CLK := #sOneStepForward;
       #sRTOneStepForward();
       #sStepForward := (NOT #sOneStepMode OR (#sOneStepMode AND #sRTOneStepForward.Q)) AND NOT #iStepPause;
       #sOneStepForward := FALSE;

       // Action only true in dedicated steps

       // Step Timer

   END_REGION

   REGION Sequence Function
       CASE #sCurrent_Step_NB OF
           #S00_INIT:
               REGION S00 INIT
                   #sCheck_Step_Condition := TRUE;
               END_REGION
           #S10_CHECK_FIXTURE_RELEASE_OPTION:
               REGION S10_CHECK_FIXTURE_RELEASE_OPTION
                   #sCheck_Step_Condition := TRUE;
               END_REGION
           #S20_AXIS_V_TO_FIXTURE_SAFE_POS_START_REQ:
               REGION S20_AXIS_V_TO_FIXTURE_SAFE_POS_START_REQ
                   #sAxisV_StartReq := NOT #iAxisV_FixtSafePos;
                   #sAxisV_PosSetPoint := LREAL_TO_REAL(#iAxisV_FixtSafePosSetPoint);
                   #sCheck_Step_Condition := TRUE;
               END_REGION
           #S30_AXIS_V_TO_FIXTURE_SAFE_POS_REACHED:
               REGION S30_AXIS_V_TO_FIXTURE_SAFE_POS_REACHED
                   #sCheck_Step_Condition := TRUE;
               END_REGION
           #S95_JOB_DONE:
               REGION S95_JOB_DONE
                   #sInterface.JobDone := TRUE;
                   #sCheck_Step_Condition := TRUE;
               END_REGION
           ELSE:
               #sInterface.Error := TRUE;
       END_CASE;
   END_REGION

   REGION Sequence Next Step Condition
       IF #sCheck_Step_Condition THEN
           CASE #sCurrent_Step_NB OF
               #S00_INIT:
                   REGION S00_INIT
                       IF #sInterface.SequenceReleased AND #iJobReq THEN
                           #sCurrent_Step_NB := #S10_CHECK_FIXTURE_RELEASE_OPTION;
                           #sInterface.SequenceRun := TRUE;
                           #sCheck_Step_Condition := FALSE;
                       ELSE
                           #sInterface.SequenceRun := FALSE;
                       END_IF;
                   END_REGION
               #S10_CHECK_FIXTURE_RELEASE_OPTION:
                   REGION S10_CHECK_FIXTURE_RELEASE_OPTION
                       IF #sInterface.SequenceReleased AND #sStepForward AND NOT "DB_LoaderOptions".Fixture.V_InitDisabled THEN
                           #sCurrent_Step_NB := #S20_AXIS_V_TO_FIXTURE_SAFE_POS_START_REQ;
                           #sCheck_Step_Condition := FALSE;
                       ELSIF #sInterface.SequenceReleased AND #sStepForward AND "DB_LoaderOptions".Fixture.V_InitDisabled THEN
                           #sCurrent_Step_NB := #S95_JOB_DONE;
                           #sCheck_Step_Condition := FALSE;
                       END_IF;
                   END_REGION
               #S20_AXIS_V_TO_FIXTURE_SAFE_POS_START_REQ:
                   REGION S20_AXIS_V_TO_FIXTURE_SAFE_POS_START_REQ
                       IF #sInterface.SequenceReleased AND #sStepForward AND (#iAxisV_Moving OR #iAxisV_FixtSafePos) THEN
                           #sCurrent_Step_NB := #S30_AXIS_V_TO_FIXTURE_SAFE_POS_REACHED;
                           #sCheck_Step_Condition := FALSE;
                       END_IF;
                   END_REGION
               #S30_AXIS_V_TO_FIXTURE_SAFE_POS_REACHED:
                   REGION S30_AXIS_V_TO_FIXTURE_SAFE_POS_REACHED
                       IF #sInterface.SequenceReleased AND #sStepForward AND NOT #sAxisV_StartReq AND #iAxisV_FixtSafePos THEN
                           #sCurrent_Step_NB := #S95_JOB_DONE;
                           #sCheck_Step_Condition := FALSE;
                       END_IF;
                   END_REGION
               #S95_JOB_DONE:
                   REGION S95_JOB_DONE
                       IF NOT #iJobReq THEN
                           #sCurrent_Step_NB := #S00_INIT;
                           #sCheck_Step_Condition := FALSE;
                           #sInterface.JobDone := FALSE;
                       END_IF;
                   END_REGION
               ELSE
                   #sInterface.Error := TRUE;
           END_CASE;
       END_IF;
   END_REGION

   REGION Outputs Update
       #oAxisV_StartReq := #sAxisV_StartReq;
       #oAxisV_PosSetPoint := #sAxisV_PosSetPoint;
   END_REGION

   REGION Steps - Date and Time History
       IF #sHistory.Activation THEN
           IF #sHistory.Steps[0] <> #sCurrent_Step_NB THEN
               FOR #tIndex := 98 TO 0 BY -1 DO
                   #sHistory.Steps[#tIndex + 1] := #sHistory.Steps[#tIndex];
                   #sHistory.Date_Time[#tIndex + 1] := #sHistory.Date_Time[#tIndex];
               END_FOR;
               #sHistory.Steps[0] := #sCurrent_Step_NB;
               #sHistory.Date_Time[0] := #iPLC_DateAndTime;
           END_IF;
       END_IF;
   END_REGION

   REGION Steps Text
       #StepText(iErrorCode := #sCurrent_Step_NB,
                 oErrorText => #StepText.oErrorText);
   END_REGION
END_FUNCTION_BLOCK

FUNCTION_BLOCK "FB_FixtureW_Init"   // FB78, SCL
{ S7_Optimized_Access := 'TRUE' }
// stored: AutoNumber false, MemoryReserve 100, SetENOAutomatically false
   VAR_INPUT
      iStartSeqCond : Bool;   // Start Sequence Conditions
      iJobReq : Bool;   // Job Request - From Main
      iAxisW_FixtSafePos : Bool;
      iAxisW_FixtSafePosSetPoint : LReal;
      iAxisW_Moving : Bool;   // Shuttle is moving
      iAxisW_InPos : Bool;
      iPLC_DateAndTime : DTL;
      iStepPause : Bool;
   END_VAR
   VAR_OUTPUT
      iAxisW_StartReq : Bool;
      iAxisW_PosSetPoint : Real;
   END_VAR
   VAR
      sCurrent_Step_NB : Int;   // Active Step Number
      sCheck_Step_Condition : Bool;
      sOneStepForward : Bool;
      sRTOneStepForward : R_TRIG;
      sOneStepMode { S7_SetPoint := 'True'} : Bool;
      sStepForward : Bool;
      sInterface : "UDT_SequenceInterface";
      sAxisW_StartReq : Bool;
      sAxisW_PosSetPoint : Real;
      sHistory : Struct
         Activation : Bool;
         Steps : Array[0..99] of Int;
         Date_Time : Array[0..99] of DTL;
      END_STRUCT;
      StepText : "FB_GetTextErrorCode";
   END_VAR
   VAR_TEMP
      tIndex : Int;   // Index
   END_VAR
   VAR CONSTANT
      S00_INIT : Int := 0;
      S10_CHECK_FIXTURE_RELEASE_OPTION : Int := 10;
      S20_AXIS_W_TO_FIXTURE_SAFE_POS_START_REQ : Int := 20;
      S30_AXIS_W_TO_FIXTURE_SAFE_POS_REACHED : Int := 30;
      S95_JOB_DONE : Int := 95;
   END_VAR
   // StepText.sCode_error[0].ErrorCode := 0;
   // StepText.sCode_error[1].ErrorCode := 10;
   // StepText.sCode_error[2].ErrorCode := 20;
   // StepText.sCode_error[3].ErrorCode := 30;
   // StepText.sCode_error[4].ErrorCode := 40;
   // StepText.sCode_error[5].ErrorCode := 50;
   // StepText.sCode_error[6].ErrorCode := 60;
   // StepText.sCode_error[7].ErrorCode := 70;
   // StepText.sCode_error[8].ErrorCode := 80;
   // StepText.sCode_error[9].ErrorCode := 90;
   // StepText.sCode_error[10].ErrorCode := 95;
BEGIN
   REGION Description header 
       //==================================================================================
       // POSALUX Swiss SA / (C) Copyright 2026
       //----------------------------------------------------------------------------------
       // Title: FB_FixtureW_Init
       // Comment/Function: 
       // Author: Fabien WALDT
       // Engineering: TIA Portal v20
       //----------------------------------------------------------------------------------
       // Change log table:
       // Version  | Date     | Expert in charge | Changes applied
       // ---------|----------|------------------|-----------------------------------------
       // 00.00.01 | 20260220 | WFA              | First released version
       // =================================================================================
   END_REGION

   REGION Define condition to start
       IF #iStartSeqCond THEN
           #sInterface.SequenceReleased := TRUE;
       ELSE
           // Standard sequencer controls
           #sInterface.SequenceReleased := FALSE;
           #sCurrent_Step_NB := #S00_INIT;
           #sInterface.SequenceRun := FALSE;
           #sInterface.JobDone := FALSE;
           #sCheck_Step_Condition := FALSE;

           // Dedicated sequencer controls
           #sAxisW_StartReq := FALSE;
           #sAxisW_PosSetPoint := 0.0;

           // Add specifics controls 
       END_IF;

       // Reset interface error
       IF #sInterface.Reset THEN
           #sInterface.Error := FALSE;
       END_IF;

       // Reset start when axis in position
       IF #iAxisW_InPos THEN
           #sAxisW_StartReq := FALSE;
       END_IF;

       // One step forward
       #sRTOneStepForward.CLK := #sOneStepForward;
       #sRTOneStepForward();
       #sStepForward := (NOT #sOneStepMode OR (#sOneStepMode AND #sRTOneStepForward.Q)) AND NOT #iStepPause;
       #sOneStepForward := FALSE;

       // Action only true in dedicated steps

       // Step Timer

   END_REGION

   REGION Sequence Function
       CASE #sCurrent_Step_NB OF
           #S00_INIT:
               REGION S00 INIT
                   #sCheck_Step_Condition := TRUE;
               END_REGION
           #S10_CHECK_FIXTURE_RELEASE_OPTION:
               REGION S10_CHECK_FIXTURE_RELEASE_OPTION
                   #sCheck_Step_Condition := TRUE;
               END_REGION
           #S20_AXIS_W_TO_FIXTURE_SAFE_POS_START_REQ:
               REGION S20_AXIS_W_TO_FIXTURE_SAFE_POS_START_REQ
                   #sAxisW_StartReq := NOT #iAxisW_FixtSafePos;
                   #sAxisW_PosSetPoint := LREAL_TO_REAL(#iAxisW_FixtSafePosSetPoint);
                   #sCheck_Step_Condition := TRUE;
               END_REGION
           #S30_AXIS_W_TO_FIXTURE_SAFE_POS_REACHED:
               REGION S30_AXIS_W_TO_FIXTURE_SAFE_POS_REACHED
                   #sCheck_Step_Condition := TRUE;
               END_REGION
           #S95_JOB_DONE:
               REGION S95_JOB_DONE
                   #sInterface.JobDone := TRUE;
                   #sCheck_Step_Condition := TRUE;
               END_REGION
           ELSE:
               #sInterface.Error := TRUE;
       END_CASE;
   END_REGION

   REGION Sequence Next Step Condition
       IF #sCheck_Step_Condition THEN
           CASE #sCurrent_Step_NB OF
               #S00_INIT:
                   REGION S00_INIT
                       IF #sInterface.SequenceReleased AND #iJobReq THEN
                           #sCurrent_Step_NB := #S10_CHECK_FIXTURE_RELEASE_OPTION;
                           #sInterface.SequenceRun := TRUE;
                           #sCheck_Step_Condition := FALSE;
                       ELSE
                           #sInterface.SequenceRun := FALSE;
                       END_IF;
                   END_REGION
               #S10_CHECK_FIXTURE_RELEASE_OPTION:
                   REGION S10_CHECK_FIXTURE_RELEASE_OPTION
                       IF #sInterface.SequenceReleased AND #sStepForward AND NOT "DB_LoaderOptions".Fixture.V_InitDisabled THEN
                           #sCurrent_Step_NB := #S20_AXIS_W_TO_FIXTURE_SAFE_POS_START_REQ;
                           #sCheck_Step_Condition := FALSE;
                       ELSIF #sInterface.SequenceReleased AND #sStepForward AND "DB_LoaderOptions".Fixture.V_InitDisabled THEN
                           #sCurrent_Step_NB := #S95_JOB_DONE;
                           #sCheck_Step_Condition := FALSE;
                       END_IF;
                   END_REGION
               #S20_AXIS_W_TO_FIXTURE_SAFE_POS_START_REQ:
                   REGION S20_AXIS_W_TO_FIXTURE_SAFE_POS_START_REQ
                       IF #sInterface.SequenceReleased AND #sStepForward AND (#iAxisW_Moving OR #iAxisW_FixtSafePos) THEN
                           #sCurrent_Step_NB := #S30_AXIS_W_TO_FIXTURE_SAFE_POS_REACHED;
                           #sCheck_Step_Condition := FALSE;
                       END_IF;
                   END_REGION
               #S30_AXIS_W_TO_FIXTURE_SAFE_POS_REACHED:
                   REGION S30_AXIS_W_TO_FIXTURE_SAFE_POS_REACHED
                       IF #sInterface.SequenceReleased AND #sStepForward AND NOT #sAxisW_StartReq AND #iAxisW_FixtSafePos THEN
                           #sCurrent_Step_NB := #S95_JOB_DONE;
                           #sCheck_Step_Condition := FALSE;
                       END_IF;
                   END_REGION
               #S95_JOB_DONE:
                   REGION S95_JOB_DONE
                       IF NOT #iJobReq THEN
                           #sCurrent_Step_NB := #S00_INIT;
                           #sCheck_Step_Condition := FALSE;
                           #sInterface.JobDone := FALSE;
                       END_IF;
                   END_REGION
               ELSE
                   #sInterface.Error := TRUE;
           END_CASE;
       END_IF;
   END_REGION

   REGION Outputs Update
       #iAxisW_StartReq := #sAxisW_StartReq;
       #iAxisW_PosSetPoint := #sAxisW_PosSetPoint;
   END_REGION

   REGION Steps - Date and Time History
       IF #sHistory.Activation THEN
           IF #sHistory.Steps[0] <> #sCurrent_Step_NB THEN
               FOR #tIndex := 98 TO 0 BY -1 DO
                   #sHistory.Steps[#tIndex + 1] := #sHistory.Steps[#tIndex];
                   #sHistory.Date_Time[#tIndex + 1] := #sHistory.Date_Time[#tIndex];
               END_FOR;
               #sHistory.Steps[0] := #sCurrent_Step_NB;
               #sHistory.Date_Time[0] := #iPLC_DateAndTime;
           END_IF;
       END_IF;
   END_REGION

   REGION Steps Text
       #StepText(iErrorCode := #sCurrent_Step_NB,
                 oErrorText => #StepText.oErrorText);
   END_REGION
END_FUNCTION_BLOCK

FUNCTION_BLOCK "FB_ExtraMissingPart"   // FB76, SCL
{ S7_Optimized_Access := 'TRUE' }
// stored: MemoryReserve 100, SetENOAutomatically false
   VAR
      sRT_UndrilledGripperClosedWithPart : R_TRIG;
      sRT_UndrilledGripperClosedWithoutPart { S7_SetPoint := 'True'} : R_TRIG;
      sRT_DrilledGripperClosedWithPart : R_TRIG;
      sRT_DrilledGripperClosedWithoutPart { S7_SetPoint := 'True'} : R_TRIG;
      sRT_FixturePartControlGood { S7_SetPoint := 'True'} : R_TRIG;
      sRT_FixturePartControlBad { S7_SetPoint := 'True'} : R_TRIG;
      sRT_UndrilledGripperOpen { S7_SetPoint := 'True'} : R_TRIG;
      sRT_DrilledGripperOpen { S7_SetPoint := 'True'} : R_TRIG;
      sTON_UndrilledGripperClosedWithPart { S7_SetPoint := 'True'} : TON_TIME;
      sTON_UndrilledGripperClosedWithoutPart { S7_SetPoint := 'True'} : TON_TIME;
      sTON_DrilledGripperClosedWithPart { S7_SetPoint := 'True'} : TON_TIME;
      sTON_DrilledGripperClosedWithoutPart { S7_SetPoint := 'True'} : TON_TIME;
      sTON_FixturePartControlGood { S7_SetPoint := 'True'} : TON_TIME;
      sTON_FixturePartControlBad { S7_SetPoint := 'True'} : TON_TIME;
      sTON_UndrilledGripperOpen { S7_SetPoint := 'True'} : TON_TIME;
      sTON_DrilledGripperOpen { S7_SetPoint := 'True'} : TON_TIME;
      sExtraPartUndrilledGripper { S7_SetPoint := 'True'} : Bool;
      sExtraPartDrilledGripper : Bool;
      sMissingPartUndrilledGripper { S7_SetPoint := 'True'} : Bool;
      sMissingPartDrilledGripper : Bool;
      sExtraPartFixture : Bool;
      sMissingPartFixture : Bool;
      sGlobalExtraMissing : Bool;
      sUndrilledGripperClosedWithPart : Bool;
      sUndrilledGripperClosedWithoutPart { S7_SetPoint := 'True'} : Bool;
      sDrilledGripperClosedWithPart : Bool;
      sDrilledGripperClosedWithoutPart { S7_SetPoint := 'True'} : Bool;
      sFixturePartControlGood { S7_SetPoint := 'True'} : Bool;
      sFixturePartControlBad { S7_SetPoint := 'True'} : Bool;
      sUndrilledGripperOpen { S7_SetPoint := 'True'} : Bool;
      sDrilledGripperOpen { S7_SetPoint := 'True'} : Bool;
   END_VAR
BEGIN
   REGION Description header 
       //==================================================================================
       // POSALUX Swiss SA / (C) Copyright 2026
       //----------------------------------------------------------------------------------
       // Title: 
       // Comment/Function: 
       // Author: Fabien WALDT
       // Engineering: TIA Portal v20
       //----------------------------------------------------------------------------------
       // Change log table:
       // Version  | Date     | Expert in charge | Changes applied
       // ---------|----------|------------------|-----------------------------------------
       // 00.00.01 | 20260205 | WFA              | First released version
       // =================================================================================
   END_REGION

   REGION Init
       #sExtraPartUndrilledGripper := FALSE;
       #sExtraPartDrilledGripper := FALSE;
       #sMissingPartUndrilledGripper := FALSE;
       #sMissingPartDrilledGripper := FALSE;
       #sExtraPartFixture := FALSE;
       #sMissingPartFixture := FALSE;
   END_REGION

   REGION Inputs Status
       #sTON_UndrilledGripperClosedWithPart(IN := "DB_GestionGripper".sUndrilledGripper.oStateCloseWithPart,
                                            PT := T#100ms);
       #sTON_UndrilledGripperClosedWithoutPart(IN := "DB_GestionGripper".sUndrilledGripper.oStateClose,
                                               PT := T#100ms);
       #sTON_DrilledGripperClosedWithPart(IN := "DB_GestionGripper".sDrilledGripper.oStateCloseWithPart,
                                          PT := T#100ms);
       #sTON_DrilledGripperClosedWithoutPart(IN := "DB_GestionGripper".sDrilledGripper.oStateClose,
                                             PT := T#100ms);
       #sTON_FixturePartControlGood(IN := "DB_GestionFixture".sFixturePartControl.oGoodPart,
                                    PT := T#100ms);
       #sTON_FixturePartControlBad(IN := "DB_GestionFixture".sFixturePartControl.oBadpart,
                                   PT := T#100ms);

       #sTON_UndrilledGripperOpen(IN := "DB_GestionGripper".sUndrilledGripper.oStateOpen,
                                  PT := T#100ms);
       #sTON_DrilledGripperOpen(IN := "DB_GestionGripper".sDrilledGripper.oStateOpen,
                                PT := T#100ms);

       #sRT_UndrilledGripperClosedWithPart(CLK := #sTON_UndrilledGripperClosedWithPart.Q);
       #sRT_UndrilledGripperClosedWithoutPart(CLK := #sTON_UndrilledGripperClosedWithoutPart.Q);
       #sRT_DrilledGripperClosedWithPart(CLK := #sTON_DrilledGripperClosedWithPart.Q);
       #sRT_DrilledGripperClosedWithoutPart(CLK := #sTON_DrilledGripperClosedWithoutPart.Q);
       #sRT_FixturePartControlGood(CLK := #sTON_FixturePartControlGood.Q);
       #sRT_FixturePartControlBad(CLK := #sTON_FixturePartControlBad.Q);
       #sRT_UndrilledGripperOpen(CLK := #sTON_UndrilledGripperOpen.Q);
       #sRT_DrilledGripperOpen(CLK := #sTON_DrilledGripperOpen.Q);

       #sUndrilledGripperClosedWithPart := #sTON_UndrilledGripperClosedWithPart.Q;
       #sUndrilledGripperClosedWithoutPart := #sTON_UndrilledGripperClosedWithoutPart.Q;
       #sDrilledGripperClosedWithPart := #sTON_DrilledGripperClosedWithPart.Q;
       #sDrilledGripperClosedWithoutPart := #sTON_DrilledGripperClosedWithoutPart.Q;
       #sFixturePartControlGood := #sTON_FixturePartControlGood.Q;
       #sFixturePartControlBad := #sTON_FixturePartControlBad.Q;
       #sUndrilledGripperOpen := #sTON_UndrilledGripperOpen.Q;
       #sDrilledGripperOpen := #sTON_DrilledGripperOpen.Q;

   END_REGION

   REGION Shuttle to Undrilled Gripper
       IF "LBP_ModeGroup".E_JOG THEN
           IF #sRT_UndrilledGripperClosedWithPart.Q AND NOT "DB_PartManagement".sPosition.sGripper.Undrilled.Presence.Part THEN
               "DB_PartManagement".sPosition.sGripper.Undrilled.Presence.Part := TRUE;
               "DB_PartManagement".sPosition.sGripper.Undrilled.Presence.BW := TRUE;
           ELSIF #sRT_UndrilledGripperClosedWithoutPart.Q AND "DB_PartManagement".sPosition.sGripper.Undrilled.Presence.Part THEN
               "DB_PartManagement".sPosition.sGripper.Undrilled.Presence.Part := FALSE;
               "DB_PartManagement".sPosition.sGripper.Undrilled.Presence.BW := FALSE;
           END_IF;
       ELSIF NOT "DB_WorkingModes".sDryRun THEN
           IF #sUndrilledGripperClosedWithPart AND NOT "DB_PartManagement".sPosition.sGripper.Undrilled.Presence.Part THEN
               #sExtraPartUndrilledGripper := TRUE;
               "LBP_AlarmMsgs".UserA[04].A70UUxx[25] := TRUE; // Msg 700425 "Extra Product Undrilled Gripper"
           ELSIF #sUndrilledGripperClosedWithoutPart AND "DB_PartManagement".sPosition.sGripper.Undrilled.Presence.Part THEN
               #sMissingPartUndrilledGripper := TRUE;
               "LBP_AlarmMsgs".UserA[04].A70UUxx[24] := TRUE; // Msg 700424 "Missing Product Undrilled Gripper"
           END_IF;
       END_IF;
   END_REGION

   REGION Undrilled Gripper to Fixture
       IF "LBP_ModeGroup".E_JOG THEN
           IF #sRT_FixturePartControlGood.Q AND NOT "DB_PartManagement".sPosition.sFixture.Undrilled.Presence.Part AND NOT "DB_PartManagement".sPosition.sFixture.Drilled.Presence.Part THEN
               "DB_PartManagement".sPosition.sFixture.Drilled.Presence.Part := TRUE;
               "DB_PartManagement".sPosition.sFixture.Drilled.Presence.BW := TRUE;
           ELSIF #sRT_FixturePartControlBad.Q AND ("DB_PartManagement".sPosition.sFixture.Undrilled.Presence.Part OR "DB_PartManagement".sPosition.sFixture.Drilled.Presence.Part) THEN
               "DB_PartManagement".sPosition.sFixture.Drilled.Presence.Part := FALSE;
               "DB_PartManagement".sPosition.sFixture.Drilled.Presence.BW := FALSE;
           END_IF;
       ELSIF NOT "DB_WorkingModes".sDryRun THEN
           IF #sFixturePartControlGood AND NOT "DB_PartManagement".sPosition.sFixture.Undrilled.Presence.Part AND NOT "DB_PartManagement".sPosition.sFixture.Drilled.Presence.Part THEN
               #sExtraPartFixture := TRUE;
               "LBP_AlarmMsgs".UserA[04].A70UUxx[27] := TRUE; // Msg 700427 "Extra Product Fixture"
           ELSIF #sFixturePartControlBad AND ("DB_PartManagement".sPosition.sFixture.Undrilled.Presence.Part OR "DB_PartManagement".sPosition.sFixture.Drilled.Presence.Part) THEN
               #sMissingPartFixture := TRUE;
               "LBP_AlarmMsgs".UserA[04].A70UUxx[26] := TRUE; // Msg 700426 "Missing Product Fixture"
           END_IF;
       END_IF;
   END_REGION

   REGION Fixture to Drilled Gripper
       IF "LBP_ModeGroup".E_JOG THEN
           IF #sRT_DrilledGripperClosedWithPart.Q AND NOT "DB_PartManagement".sPosition.sGripper.Drilled.Presence.Part THEN
               "DB_PartManagement".sPosition.sGripper.Drilled.Presence.Part := TRUE;
               "DB_PartManagement".sPosition.sGripper.Drilled.Presence.BW := TRUE;
           ELSIF #sRT_DrilledGripperClosedWithoutPart.Q AND "DB_PartManagement".sPosition.sGripper.Drilled.Presence.Part THEN
               "DB_PartManagement".sPosition.sGripper.Drilled.Presence.Part := FALSE;
               "DB_PartManagement".sPosition.sGripper.Drilled.Presence.BW := FALSE;
           END_IF;
       ELSIF NOT "DB_WorkingModes".sDryRun THEN
           IF #sDrilledGripperClosedWithPart AND NOT "DB_PartManagement".sPosition.sGripper.Drilled.Presence.Part THEN
               #sExtraPartDrilledGripper := TRUE;
               "LBP_AlarmMsgs".UserA[04].A70UUxx[29] := TRUE; // Msg 700429 "Extra Product Drilled Gripper"
           ELSIF #sDrilledGripperClosedWithoutPart AND "DB_PartManagement".sPosition.sGripper.Drilled.Presence.Part THEN
               #sMissingPartDrilledGripper := TRUE;
               "LBP_AlarmMsgs".UserA[04].A70UUxx[28] := TRUE; // Msg 700428 "Missing Product Drilled Gripper"
           END_IF;
       END_IF;
   END_REGION

   REGION Gripper Open
       IF "LBP_ModeGroup".E_JOG THEN
           IF #sRT_UndrilledGripperOpen.Q THEN
               "DB_PartManagement".sPosition.sGripper.Undrilled.Presence.Part := FALSE;
               "DB_PartManagement".sPosition.sGripper.Undrilled.Presence.BW := FALSE;
           END_IF;
           IF #sRT_DrilledGripperOpen.Q THEN
               "DB_PartManagement".sPosition.sGripper.Drilled.Presence.Part := FALSE;
               "DB_PartManagement".sPosition.sGripper.Drilled.Presence.BW := FALSE;
           END_IF;
       END_IF;
   END_REGION

   REGION Global Extra Missing
       #sGlobalExtraMissing :=
          #sExtraPartUndrilledGripper
       OR #sExtraPartDrilledGripper
       OR #sMissingPartUndrilledGripper 
       OR #sMissingPartDrilledGripper
       OR #sExtraPartFixture
       OR #sMissingPartFixture;
   END_REGION
END_FUNCTION_BLOCK

FUNCTION_BLOCK "FB_PrioSequence"   // FB79, SCL
{ S7_Optimized_Access := 'TRUE' }
// stored: MemoryReserve 100, SetENOAutomatically false
   VAR
      sPrio : Int;
   END_VAR
BEGIN
   REGION Description header 
       //==================================================================================
       // POSALUX Swiss SA / (C) Copyright 2026
       //----------------------------------------------------------------------------------
       // Title: 
       // Comment/Function: FB_PrioSequence
       // Author: Fabien WALDT
       // Engineering: TIA Portal v20
       //----------------------------------------------------------------------------------
       // Change log table:
       // Version  | Date     | Expert in charge | Changes applied
       // ---------|----------|------------------|-----------------------------------------
       // 00.00.01 | 20260205 | WFA              | First released version
       // =================================================================================
   END_REGION

   REGION Test Prio
       // #sPrio := 0;

       // IF "DB_LoaderShuttle1".sMain.sInterface.SequenceRun AND "DB_LoaderShuttle2".sMain.sInterface.SequenceRun THEN
       //     IF "DB_LoaderShuttle2".sMain.sCurrent_Step_NB > "DB_LoaderShuttle1".sMain.sCurrent_Step_NB THEN
       //         #sPrio := 2;
       //     ELSE
       //         #sPrio := 1;
       //     END_IF;
       // ELSIF "DB_LoaderShuttle1".sMain.sInterface.SequenceRun AND NOT "DB_LoaderShuttle2".sMain.sInterface.SequenceRun THEN
       //     #sPrio := 1;
       // ELSIF NOT "DB_LoaderShuttle1".sMain.sInterface.SequenceRun AND "DB_LoaderShuttle2".sMain.sInterface.SequenceRun THEN
       //     #sPrio := 2;
       // ELSE
       //     #sPrio := 0;
       // END_IF;
       // 
       IF "DB_HMISetting".Shuttle1Enable AND NOT "DB_HMISetting".Shuttle2Enable THEN
           #sPrio := 1;
       ELSIF "DB_HMISetting".Shuttle2Enable AND NOT "DB_HMISetting".Shuttle1Enable THEN
           #sPrio := 2;
       ELSIF "DB_HMISetting".Shuttle1Enable AND NOT "DB_HMISetting".Shuttle2Enable AND "DB_LoaderShuttle2".sMain.sCurrent_Step_NB > "DB_LoaderShuttle1".sMain.sCurrent_Step_NB THEN
           #sPrio := 2;
       ELSE
           #sPrio := 1;
       END_IF;
   END_REGION
END_FUNCTION_BLOCK

FUNCTION_BLOCK "FB_Alarms"   // FB300, SCL
{ S7_Optimized_Access := 'FALSE' }
// stored: AutoNumber false, SetENOAutomatically false
   VAR
      sAlarmsLevel0 : Bool;
      sAlarmsLevel1 : Bool;
      sAlarmsLevel2 : Bool;
      sAlarmsLevel3 : Bool;
      sAlarmsLevel4 : Bool;
      sAlarmsLevel5 : Bool;
      sAlarmsLevel6 : Bool;
      sRTBuzzer { S7_SetPoint := 'True'} : R_TRIG;
      sActiveBuzzer : Bool;
      sTableInParkPosition : Bool;
   END_VAR
   VAR_TEMP
      tIndexRID : Int;
   END_VAR
BEGIN
   REGION Description header 
       //==================================================================================
       // POSALUX Swiss SA / (C) Copyright 2024
       //----------------------------------------------------------------------------------
       // Title: Alarmes_Machine
       // Comment/Function: Alarm management block for the machine, organized by severity
       //                   levels (0 to 6).
       //                   Each level triggers specific actions. Alarms are grouped by
       //                   their levels.
       // Author: Gowsigan SRITHARAN
       // Engineering: TIA Portal v17
       //----------------------------------------------------------------------------------
       // Change log table:
       // Version  | Date     | Expert in charge | Changes applied
       // ---------|----------|------------------|------------------------------------
       // 00.00.01 | 20241206 | GSR              | First released version
       // ---------|----------|------------------|------------------------------------
       // ==================================================================================
   END_REGION
   REGION "Alarm" level 0
       // Messages
       #sAlarmsLevel0 :=
       "LBP_AlarmMsgs".UserA[00].A70UUxx[35]

       OR "LBP_AlarmMsgs".UserA[02].A70UUxx[36]

       OR "LBP_AlarmMsgs".UserA[05].A70UUxx[32]
       OR "LBP_AlarmMsgs".UserA[05].A70UUxx[33]
       OR "LBP_AlarmMsgs".UserA[05].A70UUxx[34]
       OR "LBP_AlarmMsgs".UserA[05].A70UUxx[35]
       OR "LBP_AlarmMsgs".UserA[05].A70UUxx[36]
       OR "LBP_AlarmMsgs".UserA[05].A70UUxx[37]
       OR "LBP_AlarmMsgs".UserA[05].A70UUxx[38]
       OR "LBP_AlarmMsgs".UserA[05].A70UUxx[39]
       OR "LBP_AlarmMsgs".UserA[05].A70UUxx[42]
       OR "LBP_AlarmMsgs".UserA[05].A70UUxx[48]
       OR "LBP_AlarmMsgs".UserA[05].A70UUxx[50]
       OR "LBP_AlarmMsgs".UserA[05].A70UUxx[51]

       OR "LBP_AlarmMsgs".UserA[08].A70UUxx[00]
       OR "LBP_AlarmMsgs".UserA[08].A70UUxx[41]

       OR "LBP_AlarmMsgs".ChanA[1].RID_5C02xx[00]
       OR "LBP_AlarmMsgs".ChanA[1].RID_5C02xx[01]
       OR "LBP_AlarmMsgs".ChanA[1].RID_5C02xx[02]
       OR "LBP_AlarmMsgs".ChanA[1].RID_5C02xx[03]
       OR "LBP_AlarmMsgs".ChanA[1].RID_5C02xx[04]
       OR "LBP_AlarmMsgs".ChanA[1].RID_5C02xx[05]
       OR "LBP_AlarmMsgs".ChanA[1].RID_5C02xx[06]
       OR "LBP_AlarmMsgs".ChanA[1].RID_5C02xx[07]
       OR "LBP_AlarmMsgs".ChanA[1].RID_5C02xx[08]
       OR "LBP_AlarmMsgs".ChanA[1].RID_5C02xx[09]
       OR "LBP_AlarmMsgs".ChanA[1].RID_5C02xx[10]
       OR "LBP_AlarmMsgs".ChanA[1].RID_5C02xx[11]
       OR "LBP_AlarmMsgs".ChanA[1].RID_5C02xx[12]
       OR "LBP_AlarmMsgs".ChanA[1].RID_5C02xx[13]
       OR "LBP_AlarmMsgs".ChanA[1].RID_5C02xx[14]
       OR "LBP_AlarmMsgs".ChanA[1].RID_5C02xx[15];
   END_REGION

   REGION "Alarm" level 1
       // Blinking blue light + user acknowledge
       #sAlarmsLevel1 :=
          "LBP_AlarmMsgs".UserA[00].A70UUxx[59]
       OR "LBP_AlarmMsgs".UserA[00].A70UUxx[60]
       OR "LBP_AlarmMsgs".UserA[00].A70UUxx[61]
       OR "LBP_AlarmMsgs".UserA[00].A70UUxx[62]

       OR "LBP_AlarmMsgs".UserA[03].A70UUxx[48]

       OR "LBP_AlarmMsgs".UserA[04].A70UUxx[41]
       OR "LBP_AlarmMsgs".UserA[04].A70UUxx[42]

       OR "LBP_AlarmMsgs".UserA[05].A70UUxx[43]

       OR "LBP_AlarmMsgs".UserA[06].A70UUxx[62]
       OR "LBP_AlarmMsgs".UserA[06].A70UUxx[63]

       OR "LBP_AlarmMsgs".UserA[30].A70UUxx[32]
       OR "LBP_AlarmMsgs".UserA[30].A70UUxx[33]
       OR "LBP_AlarmMsgs".UserA[30].A70UUxx[34]
       OR "LBP_AlarmMsgs".UserA[30].A70UUxx[35]
       OR "LBP_AlarmMsgs".UserA[30].A70UUxx[36]
       OR "LBP_AlarmMsgs".UserA[30].A70UUxx[37]
       OR "LBP_AlarmMsgs".UserA[30].A70UUxx[38]
       OR "LBP_AlarmMsgs".UserA[30].A70UUxx[39]
       OR "LBP_AlarmMsgs".UserA[30].A70UUxx[10]
       OR "LBP_AlarmMsgs".UserA[30].A70UUxx[41]
       OR "LBP_AlarmMsgs".UserA[30].A70UUxx[42]
       OR "LBP_AlarmMsgs".UserA[30].A70UUxx[43]
       OR "LBP_AlarmMsgs".UserA[30].A70UUxx[44]
       OR "LBP_AlarmMsgs".UserA[30].A70UUxx[45]
       OR "LBP_AlarmMsgs".UserA[30].A70UUxx[46]
       OR "LBP_AlarmMsgs".UserA[30].A70UUxx[47];
   END_REGION

   REGION "Alarm" level 2
       // blinking blue light and red beacon + user acknowledge
       #sAlarmsLevel2 :=
       "LBP_AlarmMsgs".UserA[00].A70UUxx[55]
       OR "LBP_AlarmMsgs".UserA[00].A70UUxx[63]

       OR "LBP_AlarmMsgs".UserA[04].A70UUxx[03]
       OR "LBP_AlarmMsgs".UserA[04].A70UUxx[04]
       OR "LBP_AlarmMsgs".UserA[04].A70UUxx[05]
       OR "LBP_AlarmMsgs".UserA[04].A70UUxx[06]
       OR "LBP_AlarmMsgs".UserA[04].A70UUxx[20]
       OR "LBP_AlarmMsgs".UserA[04].A70UUxx[21]
       OR "LBP_AlarmMsgs".UserA[04].A70UUxx[22]
       OR "LBP_AlarmMsgs".UserA[04].A70UUxx[23]

       OR "LBP_AlarmMsgs".UserA[05].A70UUxx[08]
       OR "LBP_AlarmMsgs".UserA[05].A70UUxx[09]
       OR "LBP_AlarmMsgs".UserA[05].A70UUxx[10]
       OR "LBP_AlarmMsgs".UserA[05].A70UUxx[11]
       OR "LBP_AlarmMsgs".UserA[05].A70UUxx[12]

       OR "LBP_AlarmMsgs".UserA[06].A70UUxx[52]
       OR "LBP_AlarmMsgs".UserA[06].A70UUxx[53]

       OR "LBP_AlarmMsgs".UserA[07].A70UUxx[00]
       OR "LBP_AlarmMsgs".UserA[07].A70UUxx[01]
       OR "LBP_AlarmMsgs".UserA[07].A70UUxx[02]
       OR "LBP_AlarmMsgs".UserA[07].A70UUxx[03]
       OR "LBP_AlarmMsgs".UserA[07].A70UUxx[04]
       OR "LBP_AlarmMsgs".UserA[07].A70UUxx[05]
       OR "LBP_AlarmMsgs".UserA[07].A70UUxx[06]
       OR "LBP_AlarmMsgs".UserA[07].A70UUxx[07]
       OR "LBP_AlarmMsgs".UserA[07].A70UUxx[08]
       OR "LBP_AlarmMsgs".UserA[07].A70UUxx[09]
       OR "LBP_AlarmMsgs".UserA[07].A70UUxx[10]
       OR "LBP_AlarmMsgs".UserA[07].A70UUxx[11]
       OR "LBP_AlarmMsgs".UserA[07].A70UUxx[40]
       OR "LBP_AlarmMsgs".UserA[07].A70UUxx[41]
       OR "LBP_AlarmMsgs".UserA[07].A70UUxx[42]
       OR "LBP_AlarmMsgs".UserA[07].A70UUxx[43]
       OR "LBP_AlarmMsgs".UserA[07].A70UUxx[44]
       OR "LBP_AlarmMsgs".UserA[07].A70UUxx[45]
       OR "LBP_AlarmMsgs".UserA[07].A70UUxx[46]
       OR "LBP_AlarmMsgs".UserA[07].A70UUxx[47]
       OR "LBP_AlarmMsgs".UserA[07].A70UUxx[48]
       OR "LBP_AlarmMsgs".UserA[07].A70UUxx[49]
       OR "LBP_AlarmMsgs".UserA[07].A70UUxx[50]
       OR "LBP_AlarmMsgs".UserA[07].A70UUxx[51]
       OR "LBP_AlarmMsgs".UserA[07].A70UUxx[52]
       OR "LBP_AlarmMsgs".UserA[07].A70UUxx[53]
       OR "LBP_AlarmMsgs".UserA[07].A70UUxx[54]
       OR "LBP_AlarmMsgs".UserA[07].A70UUxx[55]
       OR "LBP_AlarmMsgs".UserA[07].A70UUxx[56]
       OR "LBP_AlarmMsgs".UserA[07].A70UUxx[57]
       OR "LBP_AlarmMsgs".UserA[07].A70UUxx[58]
       OR "LBP_AlarmMsgs".UserA[07].A70UUxx[59]
       OR "LBP_AlarmMsgs".UserA[07].A70UUxx[60]
       OR "LBP_AlarmMsgs".UserA[07].A70UUxx[61]

       OR "LBP_AlarmMsgs".UserA[30].A70UUxx[00]
       OR "LBP_AlarmMsgs".UserA[30].A70UUxx[01]
       OR "LBP_AlarmMsgs".UserA[30].A70UUxx[02]
       OR "LBP_AlarmMsgs".UserA[30].A70UUxx[03]
       OR "LBP_AlarmMsgs".UserA[30].A70UUxx[04]
       OR "LBP_AlarmMsgs".UserA[30].A70UUxx[05]
       OR "LBP_AlarmMsgs".UserA[30].A70UUxx[06]
       OR "LBP_AlarmMsgs".UserA[30].A70UUxx[07]
       OR "LBP_AlarmMsgs".UserA[30].A70UUxx[08]
       OR "LBP_AlarmMsgs".UserA[30].A70UUxx[09]
       OR "LBP_AlarmMsgs".UserA[30].A70UUxx[10]
       OR "LBP_AlarmMsgs".UserA[30].A70UUxx[11]
       OR "LBP_AlarmMsgs".UserA[30].A70UUxx[12]
       OR "LBP_AlarmMsgs".UserA[30].A70UUxx[13]
       OR "LBP_AlarmMsgs".UserA[30].A70UUxx[14]
       OR "LBP_AlarmMsgs".UserA[30].A70UUxx[15];
   END_REGION

   REGION "Alarm" level 3
       // blinking blue light and red beacon + stop program at next step + user acknowledge
       #sAlarmsLevel3 :=
       "LBP_AlarmMsgs".UserA[00].A70UUxx[06]
       OR "LBP_AlarmMsgs".UserA[00].A70UUxx[07]
       OR "LBP_AlarmMsgs".UserA[00].A70UUxx[08]
       OR "LBP_AlarmMsgs".UserA[00].A70UUxx[14]
       OR "LBP_AlarmMsgs".UserA[00].A70UUxx[15]

       OR "LBP_AlarmMsgs".UserA[01].A70UUxx[03]
       OR "LBP_AlarmMsgs".UserA[01].A70UUxx[04]
       OR "LBP_AlarmMsgs".UserA[01].A70UUxx[05]
       OR "LBP_AlarmMsgs".UserA[01].A70UUxx[06]
       OR "LBP_AlarmMsgs".UserA[01].A70UUxx[07]
       OR "LBP_AlarmMsgs".UserA[01].A70UUxx[08]
       OR "LBP_AlarmMsgs".UserA[01].A70UUxx[09]
       OR "LBP_AlarmMsgs".UserA[01].A70UUxx[10]
       OR "LBP_AlarmMsgs".UserA[01].A70UUxx[11]
       OR "LBP_AlarmMsgs".UserA[01].A70UUxx[12]
       OR "LBP_AlarmMsgs".UserA[01].A70UUxx[13]
       OR "LBP_AlarmMsgs".UserA[01].A70UUxx[14]
       OR "LBP_AlarmMsgs".UserA[01].A70UUxx[15]
       OR "LBP_AlarmMsgs".UserA[01].A70UUxx[20]

       OR "LBP_AlarmMsgs".UserA[02].A70UUxx[00]
       OR "LBP_AlarmMsgs".UserA[02].A70UUxx[01]
       OR "LBP_AlarmMsgs".UserA[02].A70UUxx[02]
       OR "LBP_AlarmMsgs".UserA[02].A70UUxx[04]
       OR "LBP_AlarmMsgs".UserA[02].A70UUxx[05]
       OR "LBP_AlarmMsgs".UserA[02].A70UUxx[06]
       //   OR "LBP_AlarmMsgs".UserA[02].A70UUxx[07]
       //   OR "LBP_AlarmMsgs".UserA[02].A70UUxx[08]
       //   OR "LBP_AlarmMsgs".UserA[02].A70UUxx[09]
       //   OR "LBP_AlarmMsgs".UserA[02].A70UUxx[10]
       //   OR "LBP_AlarmMsgs".UserA[02].A70UUxx[11]
       //   OR "LBP_AlarmMsgs".UserA[02].A70UUxx[12]
       // OR "LBP_AlarmMsgs".UserA[02].A70UUxx[18]
       OR "LBP_AlarmMsgs".UserA[02].A70UUxx[19]
       OR "LBP_AlarmMsgs".UserA[02].A70UUxx[20]
       OR "LBP_AlarmMsgs".UserA[02].A70UUxx[21]
       OR "LBP_AlarmMsgs".UserA[02].A70UUxx[22]

       OR "LBP_AlarmMsgs".UserA[03].A70UUxx[15]
       OR "LBP_AlarmMsgs".UserA[03].A70UUxx[16]
       OR "LBP_AlarmMsgs".UserA[03].A70UUxx[17]
       OR "LBP_AlarmMsgs".UserA[03].A70UUxx[18]
       OR "LBP_AlarmMsgs".UserA[03].A70UUxx[19]
       OR "LBP_AlarmMsgs".UserA[03].A70UUxx[20]
       OR "LBP_AlarmMsgs".UserA[03].A70UUxx[21]
       OR "LBP_AlarmMsgs".UserA[03].A70UUxx[22]
       OR "LBP_AlarmMsgs".UserA[03].A70UUxx[23]
       OR "LBP_AlarmMsgs".UserA[03].A70UUxx[24]
       OR "LBP_AlarmMsgs".UserA[03].A70UUxx[25]
       OR "LBP_AlarmMsgs".UserA[03].A70UUxx[26]
       OR "LBP_AlarmMsgs".UserA[03].A70UUxx[27]
       OR "LBP_AlarmMsgs".UserA[03].A70UUxx[28]
     //  OR "LBP_AlarmMsgs".UserA[03].A70UUxx[29] WFA Msg défaut BW Loader, pas d'acquit nécéssaire

       OR "LBP_AlarmMsgs".UserA[04].A70UUxx[09]
       OR "LBP_AlarmMsgs".UserA[04].A70UUxx[10]
       OR "LBP_AlarmMsgs".UserA[04].A70UUxx[24]
       OR "LBP_AlarmMsgs".UserA[04].A70UUxx[25]
       OR "LBP_AlarmMsgs".UserA[04].A70UUxx[26]
       OR "LBP_AlarmMsgs".UserA[04].A70UUxx[27]
       OR "LBP_AlarmMsgs".UserA[04].A70UUxx[28]
       OR "LBP_AlarmMsgs".UserA[04].A70UUxx[29]

       OR "LBP_AlarmMsgs".UserA[06].A70UUxx[04]
       OR "LBP_AlarmMsgs".UserA[06].A70UUxx[05]
       OR "LBP_AlarmMsgs".UserA[06].A70UUxx[06]
       OR "LBP_AlarmMsgs".UserA[06].A70UUxx[07]
       OR "LBP_AlarmMsgs".UserA[06].A70UUxx[08]
    //   OR "LBP_AlarmMsgs".UserA[06].A70UUxx[09]
       OR "LBP_AlarmMsgs".UserA[06].A70UUxx[10]
     //  OR "LBP_AlarmMsgs".UserA[06].A70UUxx[11]
       OR "LBP_AlarmMsgs".UserA[06].A70UUxx[40]
       OR "LBP_AlarmMsgs".UserA[06].A70UUxx[41]
       OR "LBP_AlarmMsgs".UserA[06].A70UUxx[50]
     //  OR "LBP_AlarmMsgs".UserA[06].A70UUxx[51]
       OR "LBP_AlarmMsgs".UserA[06].A70UUxx[54]
       OR "LBP_AlarmMsgs".UserA[06].A70UUxx[55]
       // OR "LBP_AlarmMsgs".UserA[06].A70UUxx[56]
       OR "LBP_AlarmMsgs".UserA[06].A70UUxx[57]
       //  OR "LBP_AlarmMsgs".UserA[06].A70UUxx[58]
       OR "LBP_AlarmMsgs".UserA[06].A70UUxx[59]
       OR "LBP_AlarmMsgs".UserA[06].A70UUxx[60]
      // OR "LBP_AlarmMsgs".UserA[06].A70UUxx[61]

       // OR "LBP_AlarmMsgs".UserA[08].A70UUxx[08]
       OR "LBP_AlarmMsgs".UserA[08].A70UUxx[09]
       OR "LBP_AlarmMsgs".UserA[08].A70UUxx[10]
       OR "LBP_AlarmMsgs".UserA[08].A70UUxx[11]
       //  OR "LBP_AlarmMsgs".UserA[08].A70UUxx[12]
       OR "LBP_AlarmMsgs".UserA[08].A70UUxx[13]
       OR "LBP_AlarmMsgs".UserA[08].A70UUxx[14]
       OR "LBP_AlarmMsgs".UserA[08].A70UUxx[15]
       OR "LBP_AlarmMsgs".UserA[08].A70UUxx[16]
       OR "LBP_AlarmMsgs".UserA[08].A70UUxx[17]
       // OR "LBP_AlarmMsgs".UserA[08].A70UUxx[20]
       // OR "LBP_AlarmMsgs".UserA[08].A70UUxx[21]
       OR "LBP_AlarmMsgs".UserA[08].A70UUxx[22]
       // OR "LBP_AlarmMsgs".UserA[08].A70UUxx[23]
       OR "LBP_AlarmMsgs".UserA[08].A70UUxx[24];

   END_REGION

   REGION "Alarm" level 4
       // blinking blue light and red beacon + stop program at next step + acknowledge by reset button
       #sAlarmsLevel4 :=
          "LBP_AlarmMsgs".UserA[00].A70UUxx[02]
       OR "LBP_AlarmMsgs".UserA[00].A70UUxx[05]

       OR "LBP_AlarmMsgs".UserA[05].A70UUxx[01]
       OR "LBP_AlarmMsgs".UserA[05].A70UUxx[02]

    //   OR "LBP_AlarmMsgs".UserA[06].A70UUxx[42]
       OR "LBP_AlarmMsgs".UserA[06].A70UUxx[43]
    //   OR "LBP_AlarmMsgs".UserA[06].A70UUxx[44]
       OR "LBP_AlarmMsgs".UserA[06].A70UUxx[45]
       OR "LBP_AlarmMsgs".UserA[06].A70UUxx[46]
       OR "LBP_AlarmMsgs".UserA[06].A70UUxx[47]
     //  OR "LBP_AlarmMsgs".UserA[06].A70UUxx[48]
       OR "LBP_AlarmMsgs".UserA[06].A70UUxx[49];
   END_REGION

   REGION "Alarm" level 5
       // blinking blue light and red beacon + acknowledge by reset button + power off
       #sAlarmsLevel5 :=
          "LBP_AlarmMsgs".UserA[00].A70UUxx[03]
      // OR "LBP_AlarmMsgs".UserA[00].A70UUxx[04] WFA 20251205 

       // OR "LBP_AlarmMsgs".UserA[03].A70UUxx[30]
       // OR "LBP_AlarmMsgs".UserA[03].A70UUxx[31]

       OR "LBP_AlarmMsgs".UserA[05].A70UUxx[00]

       OR "LBP_AlarmMsgs".UserA[06].A70UUxx[00]
       OR "LBP_AlarmMsgs".UserA[06].A70UUxx[01]
     // OR "LBP_AlarmMsgs".UserA[06].A70UUxx[02] WFA 20251118 - A revoir temp min axe
       OR "LBP_AlarmMsgs".UserA[06].A70UUxx[03]
       OR "LBP_AlarmMsgs".UserA[06].A70UUxx[23]
       OR "LBP_AlarmMsgs".UserA[06].A70UUxx[25];
   END_REGION

   REGION "Alarm" level 6
       // Power off and shut down
       #sAlarmsLevel6 :=
          "LBP_AlarmMsgs".UserA[04].A70UUxx[02];
   END_REGION

   REGION Buzzer management
       IF #sRTBuzzer.Q THEN
           #sActiveBuzzer := TRUE;
       ELSIF "DB_McpKeyboardSignals".sAlarmReset.sKeySWStatus OR "MCP1_In".reset THEN
           #sActiveBuzzer := FALSE;
       END_IF;

       "DB_DigitalOutputs".sBuzzerActivation.sSWStatus :=
       #sActiveBuzzer
       OR "DB_McpKeyboardSignals".sLightTest.sKeySWStatus; //Test Lampes-LED
   END_REGION

   REGION Ack alarm level 0
       IF "DB_McpKeyboardSignals".sAlarmReset.sKeySWStatus OR "MCP1_In".reset THEN
           "LBP_AlarmMsgs".UserA[00].A70UUxx[35] := FALSE;

           "LBP_AlarmMsgs".UserA[02].A70UUxx[36] := FALSE;

           "LBP_AlarmMsgs".UserA[05].A70UUxx[32] := FALSE;
           "LBP_AlarmMsgs".UserA[05].A70UUxx[33] := FALSE;
           "LBP_AlarmMsgs".UserA[05].A70UUxx[34] := FALSE;
           "LBP_AlarmMsgs".UserA[05].A70UUxx[35] := FALSE;
           "LBP_AlarmMsgs".UserA[05].A70UUxx[36] := FALSE;
           "LBP_AlarmMsgs".UserA[05].A70UUxx[37] := FALSE;
           "LBP_AlarmMsgs".UserA[05].A70UUxx[38] := FALSE;
           "LBP_AlarmMsgs".UserA[05].A70UUxx[39] := FALSE;
           "LBP_AlarmMsgs".UserA[05].A70UUxx[42] := FALSE;
           "LBP_AlarmMsgs".UserA[05].A70UUxx[48] := FALSE;
           "LBP_AlarmMsgs".UserA[05].A70UUxx[50] := FALSE;
           "LBP_AlarmMsgs".UserA[05].A70UUxx[51] := FALSE;

           "LBP_AlarmMsgs".UserA[08].A70UUxx[00] := FALSE;
           "LBP_AlarmMsgs".UserA[08].A70UUxx[41] := FALSE;
       END_IF;
   END_REGION

   REGION Ack alarm level 1
       IF "DB_McpKeyboardSignals".sAlarmReset.sKeySWStatus OR "MCP1_In".reset THEN
           "LBP_AlarmMsgs".UserA[00].A70UUxx[59] := FALSE;
           "LBP_AlarmMsgs".UserA[00].A70UUxx[61] := FALSE;
           "LBP_AlarmMsgs".UserA[00].A70UUxx[62] := FALSE;

           "LBP_AlarmMsgs".UserA[04].A70UUxx[41] := FALSE;
           "LBP_AlarmMsgs".UserA[04].A70UUxx[42] := FALSE;

           "LBP_AlarmMsgs".UserA[05].A70UUxx[43] := FALSE;

           "LBP_AlarmMsgs".UserA[06].A70UUxx[62] := FALSE;
           "LBP_AlarmMsgs".UserA[06].A70UUxx[63] := FALSE;

           "LBP_AlarmMsgs".UserA[30].A70UUxx[32] := FALSE;
           "LBP_AlarmMsgs".UserA[30].A70UUxx[33] := FALSE;
           "LBP_AlarmMsgs".UserA[30].A70UUxx[34] := FALSE;
           "LBP_AlarmMsgs".UserA[30].A70UUxx[35] := FALSE;
           "LBP_AlarmMsgs".UserA[30].A70UUxx[36] := FALSE;
           "LBP_AlarmMsgs".UserA[30].A70UUxx[37] := FALSE;
           "LBP_AlarmMsgs".UserA[30].A70UUxx[38] := FALSE;
           "LBP_AlarmMsgs".UserA[30].A70UUxx[39] := FALSE;
           "LBP_AlarmMsgs".UserA[30].A70UUxx[10] := FALSE;
           "LBP_AlarmMsgs".UserA[30].A70UUxx[41] := FALSE;
           "LBP_AlarmMsgs".UserA[30].A70UUxx[42] := FALSE;
           "LBP_AlarmMsgs".UserA[30].A70UUxx[43] := FALSE;
           "LBP_AlarmMsgs".UserA[30].A70UUxx[44] := FALSE;
           "LBP_AlarmMsgs".UserA[30].A70UUxx[45] := FALSE;
           "LBP_AlarmMsgs".UserA[30].A70UUxx[46] := FALSE;
           "LBP_AlarmMsgs".UserA[30].A70UUxx[47] := FALSE;
       END_IF;
   END_REGION

   REGION Ack alarm level 2
       IF "DB_McpKeyboardSignals".sAlarmReset.sKeySWStatus OR "MCP1_In".reset THEN
           "LBP_AlarmMsgs".UserA[00].A70UUxx[63] := FALSE;

           "LBP_AlarmMsgs".UserA[04].A70UUxx[03] := FALSE;
           "LBP_AlarmMsgs".UserA[04].A70UUxx[04] := FALSE;
           "LBP_AlarmMsgs".UserA[04].A70UUxx[05] := FALSE;
           "LBP_AlarmMsgs".UserA[04].A70UUxx[06] := FALSE;
           "LBP_AlarmMsgs".UserA[04].A70UUxx[20] := FALSE;
           "LBP_AlarmMsgs".UserA[04].A70UUxx[21] := FALSE;
           "LBP_AlarmMsgs".UserA[04].A70UUxx[22] := FALSE;
           "LBP_AlarmMsgs".UserA[04].A70UUxx[23] := FALSE;

           "LBP_AlarmMsgs".UserA[05].A70UUxx[08] := FALSE;
           "LBP_AlarmMsgs".UserA[05].A70UUxx[09] := FALSE;
           "LBP_AlarmMsgs".UserA[05].A70UUxx[10] := FALSE;
           "LBP_AlarmMsgs".UserA[05].A70UUxx[11] := FALSE;
           "LBP_AlarmMsgs".UserA[05].A70UUxx[12] := FALSE;

           "LBP_AlarmMsgs".UserA[06].A70UUxx[52] := FALSE;
           "LBP_AlarmMsgs".UserA[06].A70UUxx[53] := FALSE;

           "LBP_AlarmMsgs".UserA[07].A70UUxx[00] := FALSE;
           "LBP_AlarmMsgs".UserA[07].A70UUxx[01] := FALSE;
           "LBP_AlarmMsgs".UserA[07].A70UUxx[02] := FALSE;
           "LBP_AlarmMsgs".UserA[07].A70UUxx[03] := FALSE;
           "LBP_AlarmMsgs".UserA[07].A70UUxx[04] := FALSE;
           "LBP_AlarmMsgs".UserA[07].A70UUxx[05] := FALSE;
           "LBP_AlarmMsgs".UserA[07].A70UUxx[06] := FALSE;
           "LBP_AlarmMsgs".UserA[07].A70UUxx[07] := FALSE;
           "LBP_AlarmMsgs".UserA[07].A70UUxx[08] := FALSE;
           "LBP_AlarmMsgs".UserA[07].A70UUxx[09] := FALSE;
           "LBP_AlarmMsgs".UserA[07].A70UUxx[10] := FALSE;
           "LBP_AlarmMsgs".UserA[07].A70UUxx[11] := FALSE;
           "LBP_AlarmMsgs".UserA[07].A70UUxx[40] := FALSE;
           "LBP_AlarmMsgs".UserA[07].A70UUxx[41] := FALSE;
           "LBP_AlarmMsgs".UserA[07].A70UUxx[42] := FALSE;
           "LBP_AlarmMsgs".UserA[07].A70UUxx[43] := FALSE;
           "LBP_AlarmMsgs".UserA[07].A70UUxx[44] := FALSE;
           "LBP_AlarmMsgs".UserA[07].A70UUxx[45] := FALSE;
           "LBP_AlarmMsgs".UserA[07].A70UUxx[46] := FALSE;
           "LBP_AlarmMsgs".UserA[07].A70UUxx[47] := FALSE;
           "LBP_AlarmMsgs".UserA[07].A70UUxx[48] := FALSE;
           "LBP_AlarmMsgs".UserA[07].A70UUxx[49] := FALSE;
           "LBP_AlarmMsgs".UserA[07].A70UUxx[50] := FALSE;
           "LBP_AlarmMsgs".UserA[07].A70UUxx[51] := FALSE;
           "LBP_AlarmMsgs".UserA[07].A70UUxx[52] := FALSE;
           "LBP_AlarmMsgs".UserA[07].A70UUxx[53] := FALSE;
           "LBP_AlarmMsgs".UserA[07].A70UUxx[54] := FALSE;
           "LBP_AlarmMsgs".UserA[07].A70UUxx[55] := FALSE;
           "LBP_AlarmMsgs".UserA[07].A70UUxx[56] := FALSE;
           "LBP_AlarmMsgs".UserA[07].A70UUxx[57] := FALSE;
           "LBP_AlarmMsgs".UserA[07].A70UUxx[58] := FALSE;
           "LBP_AlarmMsgs".UserA[07].A70UUxx[59] := FALSE;
           "LBP_AlarmMsgs".UserA[07].A70UUxx[60] := FALSE;
           "LBP_AlarmMsgs".UserA[07].A70UUxx[61] := FALSE;

           "LBP_AlarmMsgs".UserA[30].A70UUxx[00] := FALSE;
           "LBP_AlarmMsgs".UserA[30].A70UUxx[01] := FALSE;
           "LBP_AlarmMsgs".UserA[30].A70UUxx[02] := FALSE;
           "LBP_AlarmMsgs".UserA[30].A70UUxx[03] := FALSE;
           "LBP_AlarmMsgs".UserA[30].A70UUxx[04] := FALSE;
           "LBP_AlarmMsgs".UserA[30].A70UUxx[05] := FALSE;
           "LBP_AlarmMsgs".UserA[30].A70UUxx[06] := FALSE;
           "LBP_AlarmMsgs".UserA[30].A70UUxx[07] := FALSE;
           "LBP_AlarmMsgs".UserA[30].A70UUxx[08] := FALSE;
           "LBP_AlarmMsgs".UserA[30].A70UUxx[09] := FALSE;
           "LBP_AlarmMsgs".UserA[30].A70UUxx[10] := FALSE;
           "LBP_AlarmMsgs".UserA[30].A70UUxx[11] := FALSE;
           "LBP_AlarmMsgs".UserA[30].A70UUxx[12] := FALSE;
           "LBP_AlarmMsgs".UserA[30].A70UUxx[13] := FALSE;
           "LBP_AlarmMsgs".UserA[30].A70UUxx[14] := FALSE;
           "LBP_AlarmMsgs".UserA[30].A70UUxx[15] := FALSE;
       END_IF;
   END_REGION

   REGION Ack alarm level 3
       IF "DB_McpKeyboardSignals".sAlarmReset.sKeySWStatus OR "MCP1_In".reset THEN
           "LBP_AlarmMsgs".UserA[00].A70UUxx[06] := FALSE;
           "LBP_AlarmMsgs".UserA[00].A70UUxx[07] := FALSE;
           "LBP_AlarmMsgs".UserA[00].A70UUxx[08] := FALSE;
           "LBP_AlarmMsgs".UserA[00].A70UUxx[14] := FALSE;
           "LBP_AlarmMsgs".UserA[00].A70UUxx[15] := FALSE;

           "LBP_AlarmMsgs".UserA[01].A70UUxx[03] := FALSE;
           "LBP_AlarmMsgs".UserA[01].A70UUxx[04] := FALSE;
           "LBP_AlarmMsgs".UserA[01].A70UUxx[05] := FALSE;
           "LBP_AlarmMsgs".UserA[01].A70UUxx[06] := FALSE;
           "LBP_AlarmMsgs".UserA[01].A70UUxx[07] := FALSE;
           "LBP_AlarmMsgs".UserA[01].A70UUxx[08] := FALSE;
           "LBP_AlarmMsgs".UserA[01].A70UUxx[09] := FALSE;
           "LBP_AlarmMsgs".UserA[01].A70UUxx[10] := FALSE;
           "LBP_AlarmMsgs".UserA[01].A70UUxx[11] := FALSE;
           "LBP_AlarmMsgs".UserA[01].A70UUxx[12] := FALSE;
           "LBP_AlarmMsgs".UserA[01].A70UUxx[13] := FALSE;
           "LBP_AlarmMsgs".UserA[01].A70UUxx[14] := FALSE;
           "LBP_AlarmMsgs".UserA[01].A70UUxx[15] := FALSE;
           "LBP_AlarmMsgs".UserA[01].A70UUxx[20] := FALSE;

           "LBP_AlarmMsgs".UserA[02].A70UUxx[00] := FALSE;
           "LBP_AlarmMsgs".UserA[02].A70UUxx[01] := FALSE;
           "LBP_AlarmMsgs".UserA[02].A70UUxx[02] := FALSE;
           "LBP_AlarmMsgs".UserA[02].A70UUxx[04] := FALSE;
           "LBP_AlarmMsgs".UserA[02].A70UUxx[05] := FALSE;
           "LBP_AlarmMsgs".UserA[02].A70UUxx[06] := FALSE;
           "LBP_AlarmMsgs".UserA[02].A70UUxx[07] := FALSE;
           "LBP_AlarmMsgs".UserA[02].A70UUxx[08] := FALSE;
           "LBP_AlarmMsgs".UserA[02].A70UUxx[09] := FALSE;
           "LBP_AlarmMsgs".UserA[02].A70UUxx[10] := FALSE;
           "LBP_AlarmMsgs".UserA[02].A70UUxx[11] := FALSE;
           "LBP_AlarmMsgs".UserA[02].A70UUxx[12] := FALSE;
           "LBP_AlarmMsgs".UserA[02].A70UUxx[18] := FALSE;
           "LBP_AlarmMsgs".UserA[02].A70UUxx[19] := FALSE;
           "LBP_AlarmMsgs".UserA[02].A70UUxx[20] := FALSE;
           "LBP_AlarmMsgs".UserA[02].A70UUxx[21] := FALSE;
           "LBP_AlarmMsgs".UserA[02].A70UUxx[22] := FALSE;

           "LBP_AlarmMsgs".UserA[03].A70UUxx[15] := FALSE;
           "LBP_AlarmMsgs".UserA[03].A70UUxx[16] := FALSE;
           "LBP_AlarmMsgs".UserA[03].A70UUxx[17] := FALSE;
           "LBP_AlarmMsgs".UserA[03].A70UUxx[18] := FALSE;
           "LBP_AlarmMsgs".UserA[03].A70UUxx[19] := FALSE;
           "LBP_AlarmMsgs".UserA[03].A70UUxx[20] := FALSE;
           "LBP_AlarmMsgs".UserA[03].A70UUxx[21] := FALSE;
           "LBP_AlarmMsgs".UserA[03].A70UUxx[22] := FALSE;
           "LBP_AlarmMsgs".UserA[03].A70UUxx[23] := FALSE;
           "LBP_AlarmMsgs".UserA[03].A70UUxx[24] := FALSE;
           "LBP_AlarmMsgs".UserA[03].A70UUxx[25] := FALSE;
           "LBP_AlarmMsgs".UserA[03].A70UUxx[26] := FALSE;
           "LBP_AlarmMsgs".UserA[03].A70UUxx[27] := FALSE;
           "LBP_AlarmMsgs".UserA[03].A70UUxx[28] := FALSE;
           "LBP_AlarmMsgs".UserA[03].A70UUxx[29] := FALSE;

           "LBP_AlarmMsgs".UserA[04].A70UUxx[09] := FALSE;
           "LBP_AlarmMsgs".UserA[04].A70UUxx[10] := FALSE;
           "LBP_AlarmMsgs".UserA[04].A70UUxx[24] := FALSE;
           "LBP_AlarmMsgs".UserA[04].A70UUxx[25] := FALSE;
           "LBP_AlarmMsgs".UserA[04].A70UUxx[26] := FALSE;
           "LBP_AlarmMsgs".UserA[04].A70UUxx[27] := FALSE;
           "LBP_AlarmMsgs".UserA[04].A70UUxx[28] := FALSE;
           "LBP_AlarmMsgs".UserA[04].A70UUxx[29] := FALSE;

           "LBP_AlarmMsgs".UserA[06].A70UUxx[04] := FALSE;
           "LBP_AlarmMsgs".UserA[06].A70UUxx[05] := FALSE;
           "LBP_AlarmMsgs".UserA[06].A70UUxx[06] := FALSE;
           "LBP_AlarmMsgs".UserA[06].A70UUxx[07] := FALSE;
           "LBP_AlarmMsgs".UserA[06].A70UUxx[08] := FALSE;
           "LBP_AlarmMsgs".UserA[06].A70UUxx[09] := FALSE;
           "LBP_AlarmMsgs".UserA[06].A70UUxx[10] := FALSE;
           "LBP_AlarmMsgs".UserA[06].A70UUxx[11] := FALSE;
           "LBP_AlarmMsgs".UserA[06].A70UUxx[40] := FALSE;
           "LBP_AlarmMsgs".UserA[06].A70UUxx[41] := FALSE;
           "LBP_AlarmMsgs".UserA[06].A70UUxx[50] := FALSE;
           "LBP_AlarmMsgs".UserA[06].A70UUxx[51] := FALSE;
           "LBP_AlarmMsgs".UserA[06].A70UUxx[54] := FALSE;
           "LBP_AlarmMsgs".UserA[06].A70UUxx[55] := FALSE;
           "LBP_AlarmMsgs".UserA[06].A70UUxx[56] := FALSE;
           "LBP_AlarmMsgs".UserA[06].A70UUxx[57] := FALSE;
           "LBP_AlarmMsgs".UserA[06].A70UUxx[58] := FALSE;
           "LBP_AlarmMsgs".UserA[06].A70UUxx[59] := FALSE;
           "LBP_AlarmMsgs".UserA[06].A70UUxx[60] := FALSE;
           "LBP_AlarmMsgs".UserA[06].A70UUxx[61] := FALSE;

           "LBP_AlarmMsgs".UserA[08].A70UUxx[08] := FALSE;
           "LBP_AlarmMsgs".UserA[08].A70UUxx[09] := FALSE;
           "LBP_AlarmMsgs".UserA[08].A70UUxx[10] := FALSE;
           "LBP_AlarmMsgs".UserA[08].A70UUxx[11] := FALSE;
           "LBP_AlarmMsgs".UserA[08].A70UUxx[12] := FALSE;
           "LBP_AlarmMsgs".UserA[08].A70UUxx[13] := FALSE;
           "LBP_AlarmMsgs".UserA[08].A70UUxx[14] := FALSE;
           "LBP_AlarmMsgs".UserA[08].A70UUxx[15] := FALSE;
           "LBP_AlarmMsgs".UserA[08].A70UUxx[16] := FALSE;
           "LBP_AlarmMsgs".UserA[08].A70UUxx[17] := FALSE;

           "LBP_AlarmMsgs".UserA[08].A70UUxx[20] := FALSE;
           "LBP_AlarmMsgs".UserA[08].A70UUxx[21] := FALSE;
           "LBP_AlarmMsgs".UserA[08].A70UUxx[22] := FALSE;
           "LBP_AlarmMsgs".UserA[08].A70UUxx[23] := FALSE;
           "LBP_AlarmMsgs".UserA[08].A70UUxx[24] := FALSE;
       END_IF;
   END_REGION

   REGION Ack alarm level 4
       IF "MCP1_In".reset THEN
           "LBP_AlarmMsgs".UserA[00].A70UUxx[02] := FALSE;
           "LBP_AlarmMsgs".UserA[00].A70UUxx[05] := FALSE;

           "LBP_AlarmMsgs".UserA[05].A70UUxx[01] := FALSE;
           "LBP_AlarmMsgs".UserA[05].A70UUxx[02] := FALSE;

           "LBP_AlarmMsgs".UserA[06].A70UUxx[42] := FALSE;
           "LBP_AlarmMsgs".UserA[06].A70UUxx[43] := FALSE;
           "LBP_AlarmMsgs".UserA[06].A70UUxx[44] := FALSE;
           "LBP_AlarmMsgs".UserA[06].A70UUxx[45] := FALSE;
           "LBP_AlarmMsgs".UserA[06].A70UUxx[46] := FALSE;
           "LBP_AlarmMsgs".UserA[06].A70UUxx[47] := FALSE;
           "LBP_AlarmMsgs".UserA[06].A70UUxx[48] := FALSE;
           "LBP_AlarmMsgs".UserA[06].A70UUxx[49] := FALSE;
       END_IF;
   END_REGION

   REGION Ack alarm level 5
       IF "MCP1_In".reset THEN
           "LBP_AlarmMsgs".UserA[00].A70UUxx[03] := FALSE;
           "LBP_AlarmMsgs".UserA[00].A70UUxx[04] := FALSE;

           "LBP_AlarmMsgs".UserA[03].A70UUxx[30] := FALSE;
           "LBP_AlarmMsgs".UserA[03].A70UUxx[31] := FALSE;

